	out_cfg ( 	OUT_23_DOH,
					para_s.DOH_Debounce_s16,
					f_100Hz_DU16,
					DOH_RESISTANCE_MIN,
					DOH_RESISTANCE_MAX );

	out_cfg ( 	OUT_24_DOH,
					para_s.DOH_Debounce_s16,
					f_100Hz_DU16,
					DOH_RESISTANCE_MIN,
					DOH_RESISTANCE_MAX );

	out_cfg ( 	OUT_25_DOH,
					para_s.DOH_Debounce_s16,
					f_100Hz_DU16,
					DOH_RESISTANCE_MIN,
					DOH_RESISTANCE_MAX );

	out_cfg ( 	OUT_26_DOH,
					para_s.DOH_Debounce_s16,
					f_100Hz_DU16,
					DOH_RESISTANCE_MIN,
					DOH_RESISTANCE_MAX );

	out_cfg ( 	OUT_27_DOH,
					para_s.DOH_Debounce_s16,
					f_100Hz_DU16,
					DOH_RESISTANCE_MIN,
					DOH_RESISTANCE_MAX );

	out_cfg ( 	OUT_28_DOH,
					para_s.DOH_Debounce_s16,
					f_100Hz_DU16,
					DOH_RESISTANCE_MIN,
					DOH_RESISTANCE_MAX );

	out_cfg ( 	OUT_29_DOH,
					para_s.DOH_Debounce_s16,
					f_100Hz_DU16,
					DOH_RESISTANCE_MIN,
					DOH_RESISTANCE_MAX );

	out_cfg ( 	OUT_30_DOH,
					para_s.DOH_Debounce_s16,
					f_100Hz_DU16,
					DOH_RESISTANCE_MIN,
					DOH_RESISTANCE_MAX );

	out_cfg ( 	OUT_31_DOH,
					para_s.DOH_Debounce_s16,
					f_100Hz_DU16,
					DOH_RESISTANCE_MIN,
					DOH_RESISTANCE_MAX );

	out_cfg ( 	OUT_32_DOH,
					para_s.DOH_Debounce_s16,
					f_100Hz_DU16,
					DOH_RESISTANCE_MIN,
					DOH_RESISTANCE_MAX );

(******************************************************************************************************)
(* Analog Output Voltage *)
(******************************************************************************************************)

IF para_s.Out_Cfg_33_s16 = PWM_MODE THEN
	out_cfg	(	OUT_33_POH,							(* PWM output close loop *)
					para_s.AOV_Debounce_s16,		(* debounce time [ms] for error detection *)
					para_s.AOC_Freq_s16, 			(* dither frequency [Hz] *)
					AOV_RESISTANCE_MIN, 				(* min resistance of solenoid for error detection [mOhm]*)
					AOV_RESISTANCE_MAX );			(* max resistance of solenoid for error detection[mOhm] *)

ELSIF para_s.Out_Cfg_33_s16 = AOV_MODE THEN
	out_cfg	(	OUT_33_AOV,							(* PWM output close loop *)
					para_s.AOV_Debounce_s16,		(* debounce time [ms] for error detection *)
					para_s.AOC_Freq_s16, 			(* dither frequency [Hz] *)
					AOV_RESISTANCE_MIN, 				(* min resistance of solenoid for error detection [mOhm]*)
					AOV_RESISTANCE_MAX );			(* max resistance of solenoid for error detection[mOhm] *)

	out_cfgPI(	OUT_33_AOV,							(*Channel*)
			      para_s.AOV_Kp_s16,				(*Kp factor*)
	      		para_s.AOV_Ki_s16 );				(*Ki factor*)
END_IF

IF para_s.Out_Cfg_34_s16 = PWM_MODE THEN
	out_cfg	(	OUT_34_POH,							(* PWM output close loop *)
					para_s.AOV_Debounce_s16,		(* debounce time [ms] for error detection *)
					para_s.AOC_Freq_s16, 			(* dither frequency [Hz] *)
					AOV_RESISTANCE_MIN, 				(* min resistance of solenoid for error detection [mOhm]*)
					AOV_RESISTANCE_MAX );			(* max resistance of solenoid for error detection[mOhm] *)

ELSIF para_s.Out_Cfg_34_s16 = AOV_MODE THEN
	out_cfg	(	OUT_34_AOV,							(* PWM output close loop *)
					para_s.AOV_Debounce_s16,		(* debounce time [ms] for error detection *)
					para_s.AOC_Freq_s16, 			(* dither frequency [Hz] *)
					AOV_RESISTANCE_MIN, 				(* min resistance of solenoid for error detection [mOhm]*)
					AOV_RESISTANCE_MAX );			(* max resistance of solenoid for error detection[mOhm] *)

	out_cfgPI(	OUT_34_AOV,							(*Channel*)
			      para_s.AOV_Kp_s16,				(*Kp factor*)
	      		para_s.AOV_Ki_s16 );				(*Ki factor*)
END_IF

IF para_s.Out_Cfg_35_s16 = PWM_MODE THEN
	out_cfg	(	OUT_35_POH,							(* PWM output close loop *)
					para_s.AOV_Debounce_s16,		(* debounce time [ms] for error detection *)
					para_s.AOC_Freq_s16, 			(* dither frequency [Hz] *)
					AOV_RESISTANCE_MIN, 				(* min resistance of solenoid for error detection [mOhm]*)
					AOV_RESISTANCE_MAX );			(* max resistance of solenoid for error detection[mOhm] *)

ELSIF para_s.Out_Cfg_35_s16 = AOV_MODE THEN
	out_cfg	(	OUT_35_AOV,							(* PWM output close loop *)
					para_s.AOV_Debounce_s16,		(* debounce time [ms] for error detection *)
					para_s.AOC_Freq_s16, 			(* dither frequency [Hz] *)
					AOV_RESISTANCE_MIN, 				(* min resistance of solenoid for error detection [mOhm]*)
					AOV_RESISTANCE_MAX );			(* max resistance of solenoid for error detection[mOhm] *)

	out_cfgPI(	OUT_35_AOV,							(*Channel*)
			      para_s.AOV_Kp_s16,				(*Kp factor*)
	      		para_s.AOV_Ki_s16 );				(*Ki factor*)
END_IF

IF para_s.Out_Cfg_36_s16 = PWM_MODE THEN
	out_cfg	(	OUT_36_POH,							(* PWM output close loop *)
					para_s.AOV_Debounce_s16,		(* debounce time [ms] for error detection *)
					para_s.AOC_Freq_s16, 			(* dither frequency [Hz] *)
					AOV_RESISTANCE_MIN, 				(* min resistance of solenoid for error detection [mOhm]*)
					AOV_RESISTANCE_MAX );			(* max resistance of solenoid for error detection[mOhm] *)

ELSIF para_s.Out_Cfg_36_s16 = AOV_MODE THEN
	out_cfg	(	OUT_36_AOV,							(* PWM output close loop *)
					para_s.AOV_Debounce_s16,		(* debounce time [ms] for error detection *)
					para_s.AOC_Freq_s16, 			(* dither frequency [Hz] *)
					AOV_RESISTANCE_MIN, 				(* min resistance of solenoid for error detection [mOhm]*)
					AOV_RESISTANCE_MAX );			(* max resistance of solenoid for error detection[mOhm] *)

	out_cfgPI(	OUT_36_AOV,							(*Channel*)
			      para_s.AOV_Kp_s16,				(*Kp factor*)
	      		para_s.AOV_Ki_s16 );				(*Ki factor*)
END_IF


(******************************************************************************************************)
(* Proportional Output Low *)
(******************************************************************************************************)
IF para_s.Out_Cfg_37_s16 = PWM_MODE THEN
	out_cfg	(	OUT_37_POL,							(* PWM output close loop *)
					para_s.POL_Debounce_s16,		(* debounce time [ms] for error detection *)
					POL_CL_DITHER_FREQUENCY, 		(* dither frequency [Hz] *)
					POL_CL_RESISTANCE_MIN, 			(* min resistance of solenoid for error detection [mOhm]*)
					POL_CL_RESISTANCE_MAX );		(* max resistance of solenoid for error detection[mOhm] *)
ELSIF para_s.Out_Cfg_37_s16 = PWM_CURRENT_MODE THEN
	out_cfg	(	OUT_37_POL_CL,						(* PWM output close loop *)
					para_s.POL_Debounce_s16,		(* debounce time [ms] for error detection *)
					POL_CL_DITHER_FREQUENCY, 		(* dither frequency [Hz] *)
					POL_CL_RESISTANCE_MIN, 			(* min resistance of solenoid for error detection [mOhm]*)
					POL_CL_RESISTANCE_MAX );		(* max resistance of solenoid for error detection[mOhm] *)

	out_cfgPI(	OUT_37_POL_CL,						(*Channel*)
			      para_s.POL_Kp_s16,				(*Kp factor*)
	      		para_s.POL_Ki_s16 );				(*Ki factor*)
END_IF

IF para_s.Out_Cfg_38_s16 = PWM_MODE THEN
	out_cfg	(	OUT_38_POL,							(* PWM output close loop *)
					para_s.POL_Debounce_s16,		(* debounce time [ms] for error detection *)
					POL_CL_DITHER_FREQUENCY, 		(* dither frequency [Hz] *)
					POL_CL_RESISTANCE_MIN, 			(* min resistance of solenoid for error detection [mOhm]*)
					POL_CL_RESISTANCE_MAX );		(* max resistance of solenoid for error detection[mOhm] *)
ELSIF para_s.Out_Cfg_38_s16 = PWM_CURRENT_MODE THEN
	out_cfg	(	OUT_38_POL_CL,						(* PWM output close loop *)
					para_s.POL_Debounce_s16,		(* debounce time [ms] for error detection *)
					POL_CL_DITHER_FREQUENCY, 		(* dither frequency [Hz] *)
					POL_CL_RESISTANCE_MIN, 			(* min resistance of solenoid for error detection [mOhm]*)
					POL_CL_RESISTANCE_MAX );		(* max resistance of solenoid for error detection[mOhm] *)

	out_cfgPI(	OUT_38_POL_CL,						(*Channel*)
			      para_s.POL_Kp_s16,				(*Kp factor*)
	      		para_s.POL_Ki_s16 );				(*Ki factor*)
END_IF

IF para_s.Out_Cfg_39_s16 = PWM_MODE THEN
	out_cfg	(	OUT_39_POL,							(* PWM output close loop *)
					para_s.POL_Debounce_s16,		(* debounce time [ms] for error detection *)
					POL_CL_DITHER_FREQUENCY, 		(* dither frequency [Hz] *)
					POL_CL_RESISTANCE_MIN, 			(* min resistance of solenoid for error detection [mOhm]*)
					POL_CL_RESISTANCE_MAX );		(* max resistance of solenoid for error detection[mOhm] *)
ELSIF para_s.Out_Cfg_39_s16 = PWM_CURRENT_MODE THEN
	out_cfg	(	OUT_39_POL_CL,						(* PWM output close loop *)
					para_s.POL_Debounce_s16,		(* debounce time [ms] for error detection *)
					POL_CL_DITHER_FREQUENCY, 		(* dither frequency [Hz] *)
					POL_CL_RESISTANCE_MIN, 			(* min resistance of solenoid for error detection [mOhm]*)
					POL_CL_RESISTANCE_MAX );		(* max resistance of solenoid for error detection[mOhm] *)

	out_cfgPI(	OUT_39_POL_CL,						(*Channel*)
			      para_s.POL_Kp_s16,				(*Kp factor*)
	      		para_s.POL_Ki_s16 );				(*Ki factor*)
END_IF

IF para_s.Out_Cfg_40_s16 = PWM_MODE THEN
	out_cfg	(	OUT_40_POL,							(* PWM output close loop *)
					para_s.POL_Debounce_s16,		(* debounce time [ms] for error detection *)
					POL_CL_DITHER_FREQUENCY, 		(* dither frequency [Hz] *)
					POL_CL_RESISTANCE_MIN, 			(* min resistance of solenoid for error detection [mOhm]*)
					POL_CL_RESISTANCE_MAX );		(* max resistance of solenoid for error detection[mOhm] *)
ELSIF para_s.Out_Cfg_40_s16 = PWM_CURRENT_MODE THEN
	out_cfg	(	OUT_40_POL_CL,						(* PWM output close loop *)
					para_s.POL_Debounce_s16,		(* debounce time [ms] for error detection *)
					POL_CL_DITHER_FREQUENCY, 		(* dither frequency [Hz] *)
					POL_CL_RESISTANCE_MIN, 			(* min resistance of solenoid for error detection [mOhm]*)
					POL_CL_RESISTANCE_MAX );		(* max resistance of solenoid for error detection[mOhm] *)

	out_cfgPI(	OUT_40_POL_CL,						(*Channel*)
			      para_s.POL_Kp_s16,				(*Kp factor*)
	      		para_s.POL_Ki_s16 );				(*Ki factor*)
END_IF

IF para_s.Out_Cfg_41_s16 = PWM_MODE THEN
	out_cfg	(	OUT_41_POL,							(* PWM output close loop *)
					para_s.POL_Debounce_s16,		(* debounce time [ms] for error detection *)
					POL_CL_DITHER_FREQUENCY, 		(* dither frequency [Hz] *)
					POL_CL_RESISTANCE_MIN, 			(* min resistance of solenoid for error detection [mOhm]*)
					POL_CL_RESISTANCE_MAX );		(* max resistance of solenoid for error detection[mOhm] *)
ELSIF para_s.Out_Cfg_41_s16 = PWM_CURRENT_MODE THEN
	out_cfg	(	OUT_41_POL_CL,						(* PWM output close loop *)
					para_s.POL_Debounce_s16,		(* debounce time [ms] for error detection *)
					POL_CL_DITHER_FREQUENCY, 		(* dither frequency [Hz] *)
					POL_CL_RESISTANCE_MIN, 			(* min resistance of solenoid for error detection [mOhm]*)
					POL_CL_RESISTANCE_MAX );		(* max resistance of solenoid for error detection[mOhm] *)

	out_cfgPI(	OUT_41_POL_CL,						(*Channel*)
			      para_s.POL_Kp_s16,				(*Kp factor*)
	      		para_s.POL_Ki_s16 );				(*Ki factor*)
END_IF

IF para_s.Out_Cfg_42_s16 = PWM_MODE THEN
	out_cfg	(	OUT_42_POL,							(* PWM output close loop *)
					para_s.POL_Debounce_s16,		(* debounce time [ms] for error detection *)
					POL_CL_DITHER_FREQUENCY, 		(* dither frequency [Hz] *)
					POL_CL_RESISTANCE_MIN, 			(* min resistance of solenoid for error detection [mOhm]*)
					POL_CL_RESISTANCE_MAX );		(* max resistance of solenoid for error detection[mOhm] *)
ELSIF para_s.Out_Cfg_42_s16 = PWM_CURRENT_MODE THEN
	out_cfg	(	OUT_42_POL_CL,						(* PWM output close loop *)
					para_s.POL_Debounce_s16,		(* debounce time [ms] for error detection *)
					POL_CL_DITHER_FREQUENCY, 		(* dither frequency [Hz] *)
					POL_CL_RESISTANCE_MIN, 			(* min resistance of solenoid for error detection [mOhm]*)
					POL_CL_RESISTANCE_MAX );		(* max resistance of solenoid for error detection[mOhm] *)

	out_cfgPI(	OUT_42_POL_CL,						(*Channel*)
			      para_s.POL_Kp_s16,				(*Kp factor*)
	      		para_s.POL_Ki_s16 );				(*Ki factor*)
END_IF

IF para_s.Out_Cfg_43_s16 = PWM_MODE THEN
	out_cfg	(	OUT_43_POL,							(* PWM output close loop *)
					para_s.POL_Debounce_s16,		(* debounce time [ms] for error detection *)
					POL_CL_DITHER_FREQUENCY, 		(* dither frequency [Hz] *)
					POL_CL_RESISTANCE_MIN, 			(* min resistance of solenoid for error detection [mOhm]*)
					POL_CL_RESISTANCE_MAX );		(* max resistance of solenoid for error detection[mOhm] *)
ELSIF para_s.Out_Cfg_43_s16 = PWM_CURRENT_MODE THEN
	out_cfg	(	OUT_43_POL_CL,						(* PWM output close loop *)
					para_s.POL_Debounce_s16,		(* debounce time [ms] for error detection *)
					POL_CL_DITHER_FREQUENCY, 		(* dither frequency [Hz] *)
					POL_CL_RESISTANCE_MIN, 			(* min resistance of solenoid for error detection [mOhm]*)
					POL_CL_RESISTANCE_MAX );		(* max resistance of solenoid for error detection[mOhm] *)

	out_cfgPI(	OUT_43_POL_CL,						(*Channel*)
			      para_s.POL_Kp_s16,				(*Kp factor*)
	      		para_s.POL_Ki_s16 );				(*Ki factor*)
END_IF

IF para_s.Out_Cfg_44_s16 = PWM_MODE THEN
	out_cfg	(	OUT_44_POL,							(* PWM output close loop *)
					para_s.POL_Debounce_s16,		(* debounce time [ms] for error detection *)
					POL_CL_DITHER_FREQUENCY, 		(* dither frequency [Hz] *)
					POL_CL_RESISTANCE_MIN, 			(* min resistance of solenoid for error detection [mOhm]*)
					POL_CL_RESISTANCE_MAX );		(* max resistance of solenoid for error detection[mOhm] *)
ELSIF para_s.Out_Cfg_44_s16 = PWM_CURRENT_MODE THEN
	out_cfg	(	OUT_44_POL_CL,						(* PWM output close loop *)
					para_s.POL_Debounce_s16,		(* debounce time [ms] for error detection *)
					POL_CL_DITHER_FREQUENCY, 		(* dither frequency [Hz] *)
					POL_CL_RESISTANCE_MIN, 			(* min resistance of solenoid for error detection [mOhm]*)
					POL_CL_RESISTANCE_MAX );		(* max resistance of solenoid for error detection[mOhm] *)

	out_cfgPI(	OUT_44_POL_CL,						(*Channel*)
			      para_s.POL_Kp_s16,				(*Kp factor*)
	      		para_s.POL_Ki_s16 );				(*Ki factor*)
END_IF

IF para_s.Out_Cfg_45_s16 = PWM_MODE THEN
	out_cfg	(	OUT_45_POL,							(* PWM output close loop *)
					para_s.POL_Debounce_s16,		(* debounce time [ms] for error detection *)
					POL_CL_DITHER_FREQUENCY, 		(* dither frequency [Hz] *)
					POL_CL_RESISTANCE_MIN, 			(* min resistance of solenoid for error detection [mOhm]*)
					POL_CL_RESISTANCE_MAX );		(* max resistance of solenoid for error detection[mOhm] *)
ELSIF para_s.Out_Cfg_45_s16 = PWM_CURRENT_MODE THEN
	out_cfg	(	OUT_45_POL_CL,						(* PWM output close loop *)
					para_s.POL_Debounce_s16,		(* debounce time [ms] for error detection *)
					POL_CL_DITHER_FREQUENCY, 		(* dither frequency [Hz] *)
					POL_CL_RESISTANCE_MIN, 			(* min resistance of solenoid for error detection [mOhm]*)
					POL_CL_RESISTANCE_MAX );		(* max resistance of solenoid for error detection[mOhm] *)

	out_cfgPI(	OUT_45_POL_CL,						(*Channel*)
			      para_s.POL_Kp_s16,				(*Kp factor*)
	      		para_s.POL_Ki_s16 );				(*Ki factor*)
END_IF

IF para_s.Out_Cfg_46_s16 = PWM_MODE THEN
	out_cfg	(	OUT_46_POL,							(* PWM output close loop *)
					para_s.POL_Debounce_s16,		(* debounce time [ms] for error detection *)
					POL_CL_DITHER_FREQUENCY, 		(* dither frequency [Hz] *)
					POL_CL_RESISTANCE_MIN, 			(* min resistance of solenoid for error detection [mOhm]*)
					POL_CL_RESISTANCE_MAX );		(* max resistance of solenoid for error detection[mOhm] *)
ELSIF para_s.Out_Cfg_46_s16 = PWM_CURRENT_MODE THEN
	out_cfg	(	OUT_46_POL_CL,						(* PWM output close loop *)
					para_s.POL_Debounce_s16,		(* debounce time [ms] for error detection *)
					POL_CL_DITHER_FREQUENCY, 		(* dither frequency [Hz] *)
					POL_CL_RESISTANCE_MIN, 			(* min resistance of solenoid for error detection [mOhm]*)
					POL_CL_RESISTANCE_MAX );		(* max resistance of solenoid for error detection[mOhm] *)

	out_cfgPI(	OUT_46_POL_CL,						(*Channel*)
			      para_s.POL_Kp_s16,				(*Kp factor*)
	      		para_s.POL_Ki_s16 );				(*Ki factor*)
END_IF


(******************************************************************************************************)
(* Analog Current Output *)
(******************************************************************************************************)

IF para_s.Out_Cfg_47_s16 = AOC_MODE THEN

	out_cfg (	OUT_47_AOC,
					para_s.AOC_Debounce_s16,
					para_s.AOC_Freq_s16,
					AOC_RESISTANCE_MIN,
					AOC_RESISTANCE_MAX);

	out_cfgPI(	OUT_47_AOC,							(*Channel*)
			      para_s.AOC_Kp_s16,				(*Kp factor*)
	      		para_s.AOC_Ki_s16 );				(*Ki factor*)
ELSIF para_s.Out_Cfg_47_s16 = AOV_MODE THEN
	out_cfg (	OUT_47_AOV,
					para_s.AOC_Debounce_s16,
					para_s.AOC_Freq_s16,
					AOC_RESISTANCE_MIN,
					AOC_RESISTANCE_MAX);

	out_cfgPI(	OUT_47_AOV,							(*Channel*)
			      para_s.AOC_Kp_s16,				(*Kp factor*)
	      		para_s.AOC_Ki_s16 );				(*Ki factor*)
END_IF

(*see API description for more explanations about the "min resistance" and "max resistance" parameters of the "out_cfg" function*)
END_ACTION
ACTION PLC_initCAN:
(*
!!! CAN1 always at 250kBaud !!!
!!! BODAS-service always on CAN1 !!!
!!! Databox No 1 and 2 are reserved by diagnosis !!!
!!! The first 20 databoxes of each CAN channel do not need a registration !!!
*)
(*can_setTxCycle(CAN_1, CAN1_MESSAGE_FREQ);*)
can_registerTxDataboxes(CAN_1, ADR(CAN_S.Data.can_TxMsg_as[1]), 42);
(*can_registerTxBuf(CAN_s.Chnl.ELOBAU_u8, ADR(CAN_s.Data.can_1_TxBuf_as[1]), 50);*)
(************************************************************************************************)
(******************** @CAN Initialization of CAN at 250kBaud ************************************)
(************************************************************************************************)

	can_cfgRxDatabox( CAN_s.Chnl.CAN_modem_u8,
							CAN_s.Box.Rx_Start_Stop_Button,
							CAN_s.Id.Rx_Start_Stop_Button,
							CAN_EXD_DU8		);


	can_cfgRxDatabox( CAN_s.Chnl.Remote_Control_u8,
							CAN_s.Box.Rx_RemoteControl_A_u16,
							CAN_s.Id.Rx_RemoteControl_A_u16,
							CAN_STD_DU8									);

	can_cfgRxDatabox( CAN_s.Chnl.Remote_Control_u8,
							CAN_s.Box.Rx_RemoteControl_B_u16,
						CAN_s.Id.Rx_RemoteControl_B_u16,
								CAN_STD_DU8									);

	can_cfgRxDatabox( CAN_s.Chnl.Remote_Control_u8,
							CAN_s.Box.Rx_RemoteControl_C_u16,
							CAN_s.Id.Rx_RemoteControl_C_u16,
							CAN_STD_DU8									);


	can_cfgRxDatabox( CAN_s.Chnl.Remote_Control_u8,
							CAN_s.Box.Rx_RemoteControl_C_u16,
							CAN_s.Id.Rx_RemoteControl_C_u16,
							CAN_STD_DU8									);

	can_cfgRxDatabox( CAN_1, 9, 16#18DA08F3, CAN_EXD_DU8);

		(*can_cfgTxDatabox(	CAN_s.Chnl.Remote_Control_u8,
								CAN_s.Box.Tx_Remote_Control_u16,
								CAN_s.Id.Tx_RemoteControl_u16,
								CAN_STD_DU8									);*)
(*END_IF*)
(***************************************************************************************************)
(***************************************************************************************************)
can_cfgRxDatabox( CAN_s.Chnl.CAN_modem_u8,
						CAN_s.Box.Rx_Modem_300,
						CAN_s.Id.Rx_Modem_300,
						CAN_EXD_DU8									);

can_cfgRxDatabox( CAN_s.Chnl.CAN_modem_u8,
						CAN_s.Box.Rx_Modem_301,
						CAN_s.Id.Rx_Modem_301,
						CAN_EXD_DU8									);


(***************************************************************************************************)

	can_cfgTxDatabox( CAN_1, 42, 16#18DAF308, CAN_EXD_DU8);

	can_cfgTxDatabox(	CAN_s.Chnl.CAN_modem_u8,
							CAN_s.Box.Tx_Modem_202,
							CAN_s.Id.Tx_Modem_202,
							CAN_EXD_DU8									);

	can_cfgTxDatabox(	CAN_s.Chnl.CAN_modem_u8,
							CAN_s.Box.Tx_Modem_203,
							CAN_s.Id.Tx_Modem_203,
							CAN_EXD_DU8									);

	can_cfgTxDatabox(	CAN_s.Chnl.CAN_modem_u8,
							CAN_s.Box.Tx_Modem_204,
							CAN_s.Id.Tx_Modem_204,
							CAN_EXD_DU8									);

	can_cfgTxDatabox(	CAN_s.Chnl.CAN_modem_u8,
							CAN_s.Box.Tx_Modem_205,
							CAN_s.Id.Tx_Modem_205,
							CAN_EXD_DU8									);

	can_cfgTxDatabox(	CAN_s.Chnl.CAN_modem_u8,
							CAN_s.Box.Tx_Modem_206,
							CAN_s.Id.Tx_Modem_206,
							CAN_EXD_DU8									);

	can_cfgTxDatabox(	CAN_s.Chnl.CAN_modem_u8,
							CAN_s.Box.Tx_Modem_207,
							CAN_s.Id.Tx_Modem_207,
							CAN_EXD_DU8									);

	can_cfgTxDatabox(	CAN_s.Chnl.CAN_modem_u8,
							CAN_s.Box.Tx_Modem_208,
							CAN_s.Id.Tx_Modem_208,
							CAN_EXD_DU8									);

	can_cfgTxDatabox(	CAN_s.Chnl.CAN_modem_u8,
							CAN_s.Box.Tx_Modem_209,
							CAN_s.Id.Tx_Modem_209,
							CAN_EXD_DU8									);

	can_cfgTxDatabox(	CAN_s.Chnl.CAN_modem_u8,
							CAN_s.Box.Tx_Modem_210,
							CAN_s.Id.Tx_Modem_210,
							CAN_EXD_DU8									);

	can_cfgTxDatabox(	CAN_s.Chnl.CAN_modem_u8,
							CAN_s.Box.Tx_Modem_211,
							CAN_s.Id.Tx_Modem_211,
							CAN_EXD_DU8									);

	can_cfgTxDatabox(	CAN_s.Chnl.CAN_modem_u8,
							CAN_s.Box.Tx_Modem_212,
							CAN_s.Id.Tx_Modem_212,
							CAN_EXD_DU8									);

	can_cfgTxDatabox(	CAN_s.Chnl.CAN_modem_u8,
							CAN_s.Box.Tx_Modem_213,
							CAN_s.Id.Tx_Modem_213,
							CAN_EXD_DU8									);

	can_cfgTxDatabox(	CAN_s.Chnl.CAN_modem_u8,
							CAN_s.Box.Tx_Modem_214,
							CAN_s.Id.Tx_Modem_214,
							CAN_EXD_DU8									);

	can_cfgTxDatabox(	CAN_s.Chnl.CAN_modem_u8,
							CAN_s.Box.Tx_Modem_215,
							CAN_s.Id.Tx_Modem_215,
							CAN_EXD_DU8									);

	can_cfgTxDatabox(	CAN_s.Chnl.CAN_modem_u8,
							CAN_s.Box.Tx_Modem_216,
							CAN_s.Id.Tx_Modem_216,
							CAN_EXD_DU8									);

	can_cfgTxDatabox(	CAN_s.Chnl.CAN_modem_u8,
							CAN_s.Box.Tx_MI3_220,
							CAN_s.Id.Tx_MI3_220,
							CAN_EXD_DU8									);

	can_cfgTxDatabox(	CAN_s.Chnl.CAN_modem_u8,
							CAN_s.Box.Tx_MI3_221,
							CAN_s.Id.Tx_MI3_221,
							CAN_EXD_DU8									);

	can_cfgTxDatabox(	CAN_s.Chnl.CAN_modem_u8,
							CAN_s.Box.Tx_Modem_303,
							CAN_s.Id.Tx_Modem_303,
							CAN_EXD_DU8									);

	can_cfgTxDatabox(	CAN_s.Chnl.CAN_modem_u8,
							CAN_s.Box.Tx_Modem_304,
							CAN_s.Id.Tx_Modem_304,
							CAN_EXD_DU8									);

	can_cfgTxDatabox(	CAN_s.Chnl.CAN_modem_u8,
							CAN_s.Box.Tx_Modem_305,
							CAN_s.Id.Tx_Modem_305,
							CAN_EXD_DU8									);

	can_cfgTxDatabox(	CAN_s.Chnl.CAN_modem_u8,
							CAN_s.Box.Tx_Modem_306,
							CAN_s.Id.Tx_Modem_306,
							CAN_EXD_DU8									);

	can_cfgTxDatabox(	CAN_s.Chnl.CAN_modem_u8,
							CAN_s.Box.Tx_Modem_307,
							CAN_s.Id.Tx_Modem_307,
							CAN_EXD_DU8									);

	can_cfgTxDatabox(	CAN_s.Chnl.CAN_modem_u8,
							CAN_s.Box.Tx_Modem_308,
							CAN_s.Id.Tx_Modem_308,
							CAN_EXD_DU8									);

	can_cfgTxDatabox(	CAN_s.Chnl.CAN_modem_u8,
							CAN_s.Box.Tx_Modem_309,
							CAN_s.Id.Tx_Modem_309,
							CAN_EXD_DU8									);

	can_cfgTxDatabox(	CAN_s.Chnl.CAN_modem_u8,
							CAN_s.Box.Tx_Modem_310,
							CAN_s.Id.Tx_Modem_310,
							CAN_EXD_DU8									);

	can_cfgTxDatabox(	CAN_s.Chnl.CAN_modem_u8,
							CAN_s.Box.Tx_Modem_311,
							CAN_s.Id.Tx_Modem_311,
							CAN_EXD_DU8									);

	can_cfgTxDatabox(	CAN_s.Chnl.CAN_modem_u8,
							CAN_s.Box.Tx_Modem_401,
							CAN_s.Id.Tx_Modem_401,
							CAN_EXD_DU8									);

	can_cfgTxDatabox(	CAN_s.Chnl.CAN_modem_u8,
							CAN_s.Box.Tx_Modem_402,
							CAN_s.Id.Tx_Modem_402,
							CAN_EXD_DU8									);

	can_cfgTxDatabox(	CAN_s.Chnl.CAN_modem_u8,
							CAN_s.Box.Tx_Modem_405,
							CAN_s.Id.Tx_Modem_405,
							CAN_EXD_DU8									);

	can_cfgTxDatabox(	CAN_s.Chnl.CAN_modem_u8,
							CAN_s.Box.Tx_Modem_406,
							CAN_s.Id.Tx_Modem_406,
							CAN_EXD_DU8									);

(*IF typeIndModule = DM_01 AND typeDieselSpSource	= CAN_TSC1 THEN*)
	can_cfgTxDatabox(	CAN_s.Chnl.CAN_modem_u8,
							CAN_s.Box.Tx_DM1_Diesel,
							CAN_s.Id.Tx_DM1_Diesel,
							CAN_EXD_DU8									);

	can_cfgTxDatabox(	CAN_s.Chnl.CAN_modem_u8,
							CAN_s.Box.Tx_DM2_Diesel,
							CAN_s.Id.Tx_DM2_Diesel,
							CAN_EXD_DU8									);

	can_cfgTxDatabox(	CAN_1,
							3,
							16#101,
							CAN_STD_DU8	);

(* Start CAN channel *)
can_init(CAN_1,	BAUD_250K);

	can_cfgTxDatabox(	CAN_2,
							3,
							16#102,
							CAN_STD_DU8	);

can_init(CAN_2,	BAUD_250K);

	can_cfgTxDatabox(	CAN_3,
							3,
							16#103,
							CAN_STD_DU8	);

can_init(CAN_3,	BAUD_250K);

	can_cfgTxDatabox(	CAN_4,
							3,
							16#104,
							CAN_STD_DU8	);

can_init(CAN_4,	BAUD_250K);
END_ACTION
ACTION PLC_initJ1939:
(************************************************************************************************)
(******************** @CAN Initialization of the databoxes to transmit **************************)
(************************************************************************************************)
(*CAN EASY functions are used. Be aware only 20 databoxes are supported*)
(*************************************************************************************************)
(********************************* Init J1939 - from API documentation ***************************)
(*************************************************************************************************)
 (* register can rx/tx buffers *)
  (*can_registerTxBuf(CAN_1, ADR(can1_tx_buf), 30); *)     (* not needed here !!! *)
  (*can_registerRxBuf(CAN_1, ADR(can1_rx_buf), 30); *)

  (* register j1939 rx/tx message boxes:
This FUNCTION registers memory FOR j1939 receive databoxes AND therefore defines the maximal number 
OF usable J1939 receive databoxes.

Remarks:
This function must be called once during the configuration of the J1939 communication stack before 
j1939_initComm(). After the execution of this function, each j1939 receive databox has to be 
initialized with j1939_initRxDatabox() before using. The meaning of this function is similar to 
the system function can_registerRxDataboxes().    *)

j1939_registerRxDataboxes( ADR(J1939_s.Data.j1939_RxMsg_as[1]), 8);
j1939_registerTxDataboxes( ADR(J1939_s.Data.j1939_TxMsg_as[1]), 20);

  (* Define j1939 receive messages within the j1939 RX databoxes: *)
  j1939_initRxDatabox(	J1939_s.Box.Rx_EEC1_u16,
								J1939_s.PGN.EEC1,
								J1939_s.SOURCE_ADRESS,
								J1939_s.TIMEOUT.EEC1,
								J1939_s.TIMEOUT.EEC1,
								J1939_s.Length.J1939_STD_MSG_LEN,
								ADR(J1939_s.Data.RxEEC1_au8[1]),
								J1939_s.DISABLE_CALLBACK				);

  j1939_initRxDatabox(	J1939_s.Box.Rx_ET1_u16,
								J1939_s.PGN.ET1_u32,
								J1939_s.SOURCE_ADRESS,
								J1939_s.TIMEOUT.ET1_u16,
								J1939_s.TIMEOUT.ET1_u16,
								J1939_s.Length.J1939_STD_MSG_LEN,
								ADR(J1939_s.Data.RxET1_au8[1]),
								J1939_s.DISABLE_CALLBACK				);

  j1939_initRxDatabox(	J1939_s.Box.Rx_EFL_u16,
								J1939_s.PGN.EFL_u32,
								J1939_s.SOURCE_ADRESS,
								J1939_s.TIMEOUT.EFL_u16,
								J1939_s.TIMEOUT.EFL_u16,
								J1939_s.Length.J1939_STD_MSG_LEN,
								ADR(J1939_s.Data.RxEFL_au8[1]),
								J1939_s.DISABLE_CALLBACK				);

  j1939_initRxDatabox(	J1939_s.Box.Rx_IC1_u16,
								J1939_s.PGN.IC1_u32,
								J1939_s.SOURCE_ADRESS,
								J1939_s.TIMEOUT.IC1_u16,
								J1939_s.TIMEOUT.IC1_u16,
								J1939_s.Length.J1939_STD_MSG_LEN,
								ADR(J1939_s.Data.RxIC1_au8[1]),
								J1939_s.DISABLE_CALLBACK				);

  j1939_initRxDatabox(	J1939_s.Box.Rx_DD_u16,
								J1939_s.PGN.DD,
								3,	(* Посылка не от двигателя *)
								J1939_s.TIMEOUT.DD_timeout,
								J1939_s.TIMEOUT.DD_timeout,
								J1939_s.Length.J1939_STD_MSG_LEN,
								ADR(J1939_s.Data.RxDD_au8[1]),
								J1939_s.DISABLE_CALLBACK				);

  (* Define j1939 receive messages within the j1939 RX databoxes: *)
  (*j1939_initRxDatabox(	J1939_s.Box.Rx_EEC2_u16,
								J1939_s.PGN.EEC2,
								J1939_s.SOURCE_ADRESS,
								J1939_s.TIMEOUT.EEC2,
								J1939_s.TIMEOUT.EEC2,
								J1939_s.Length.J1939_STD_MSG_LEN,
								ADR(J1939_s.Data.RxEEC2_au8[1]),
								J1939_s.DISABLE_CALLBACK				);

  (* Define j1939 receive messages within the j1939 RX databoxes: *)
  j1939_initRxDatabox(	J1939_s.Box.Rx_EEC3_u16,
								J1939_s.PGN.EEC3,
								J1939_s.SOURCE_ADRESS,
								J1939_s.TIMEOUT.EEC3,
								J1939_s.TIMEOUT.EEC3,
								J1939_s.Length.J1939_STD_MSG_LEN,
								ADR(J1939_s.Data.RxEEC3_au8[1]),
								J1939_s.DISABLE_CALLBACK				);*)

(*Tx***************************************************************************************************************)
(*********** 00 ************************************************************************)
	j1939_initTxDatabox(	J1939_s.Box.Tx_TF_u16,
   							J1939_s.PGN.TF_u32,
   							J1939_s.Length.PRIOR_DEFAULT, 		(* Prioritet *)
   							J1939_s.Length.CYCLE_DEFAULT,
   							J1939_s.Length.OFFSET_10,				(* offset *)
   							J1939_s.Length.J1939_STD_MSG_LEN, 	(* Length, byte *)
   							ADR( J1939_s.Data.TxTF_au8[1]),
   							J1939_s.DISABLE_CALLBACK				);
(*********** 01 ************************************************************************)
	j1939_initTxDatabox(	J1939_s.Box.Tx_ETC2_u16,
   							J1939_s.PGN.ETC2_u32,
   							J1939_s.Length.PRIOR_DEFAULT, 		(* Prioritet *)
   							J1939_s.Length.CYCLE_DEFAULT,
   							J1939_s.Length.OFFSET_10, 				(* offset *)
   							J1939_s.Length.J1939_STD_MSG_LEN, 	(* Length, byte *)
   							ADR( J1939_s.Data.TxETC2_au8[1]),
   							J1939_s.DISABLE_CALLBACK				);
(*********** 02 ************************************************************************)

(*********** 03 ************************************************************************)
	(*j1939_initTxDatabox(	J1939_S.Box.Tx_TFAC_u16,
								J1939_s.PGN.TFAC,
								J1939_s.Length.PRIOR_DEFAULT,
								J1939_s.Length.CYCLE_TFAC,
								J1939_s.Length.OFFSET_0,
								J1939_s.Length.J1939_STD_MSG_LEN,
								ADR(J1939_s.Data.TxTFAC_au8[1]),
								J1939_s.DISABLE_CALLBACK				);*)
(*********** 04 ************************************************************************)
	(*j1939_initTxDatabox(	J1939_s.Box.Tx_ETC2_u16,
   							J1939_s.PGN.ETC2_u32,
   							J1939_s.Length.PRIOR_DEFAULT,
								J1939_s.Length.CYCLE_DEFAULT,
								J1939_s.Length.OFFSET_0,
								J1939_s.Length.J1939_STD_MSG_LEN,
   							ADR( J1939_s.Data.TxETC2_au8[1]),
   							J1939_s.DISABLE_CALLBACK				);*)
(*********** 05 ************************************************************************)
	j1939_initTxDatabox(	J1939_s.Box.Tx_BJM1,
  	 							J1939_s.PGN.BJM1,
   							J1939_s.Length.PRIOR_DEFAULT,
								J1939_s.Length.CYCLE_LOCARUS,
								J1939_s.Length.OFFSET_10,
								J1939_s.Length.J1939_STD_MSG_LEN,
   							ADR( J1939_s.Data.TxBJM1[1]),
   							J1939_s.DISABLE_CALLBACK				);
(*********** 06 ************************************************************************)
	j1939_initTxDatabox(	J1939_s.Box.Tx_AV00MF,
  	 							J1939_s.PGN.AV00MF,
   							J1939_s.Length.PRIOR_DEFAULT,
								J1939_s.Length.CYCLE_LOCARUS,
								J1939_s.Length.OFFSET_20,
								J1939_s.Length.J1939_STD_MSG_LEN,
   							ADR( J1939_s.Data.TxAV00MF[1]),
   							J1939_s.DISABLE_CALLBACK				);
(*********** 07 ************************************************************************)
	j1939_initTxDatabox(	J1939_s.Box.Tx_AV01MF,
  	 							J1939_s.PGN.AV01MF,
   							J1939_s.Length.PRIOR_DEFAULT,
								J1939_s.Length.CYCLE_LOCARUS,
								J1939_s.Length.OFFSET_20,
								J1939_s.Length.J1939_STD_MSG_LEN,
   							ADR( J1939_s.Data.TxAV01MF[1]),
   							J1939_s.DISABLE_CALLBACK				);
(*********** 08 ************************************************************************)
	j1939_initTxDatabox(	J1939_s.Box.Tx_VF,
  	 							J1939_s.PGN.VF,
   							J1939_s.Length.PRIOR_DEFAULT,
								J1939_s.Length.CYCLE_LOCARUS,
								J1939_s.Length.OFFSET_0,
								J1939_s.Length.J1939_STD_MSG_LEN,
   							ADR( J1939_s.Data.TxVF[1]),
   							J1939_s.DISABLE_CALLBACK				);
(*********** 09 ************************************************************************)
	j1939_initTxDatabox(	J1939_s.Box.Tx_TRF2,
  	 							J1939_s.PGN.TRF2,
   							J1939_s.Length.PRIOR_DEFAULT,
								J1939_s.Length.CYCLE_LOCARUS,
								J1939_s.Length.OFFSET_0,
								J1939_s.Length.J1939_STD_MSG_LEN,
   							ADR( J1939_s.Data.TxTRF2[1]),
   							J1939_s.DISABLE_CALLBACK				);
(*********** 10 ************************************************************************)
	j1939_initTxDatabox(	J1939_s.Box.Tx_MP,
  	 							J1939_s.PGN.MP,
   							J1939_s.Length.PRIOR_DEFAULT,
								J1939_s.Length.CYCLE_LOCARUS,
								J1939_s.Length.OFFSET_0,
								J1939_s.Length.J1939_STD_MSG_LEN,
   							ADR( J1939_s.Data.TxMP[1]),
   							J1939_s.DISABLE_CALLBACK				);
(*********** 11 ************************************************************************)
	j1939_initTxDatabox(	J1939_s.Box.Tx_HOURS,
  	 							J1939_s.PGN.HOURS,
   							J1939_s.Length.PRIOR_DEFAULT,
								J1939_s.Length.CYCLE_LOCARUS,
								J1939_s.Length.OFFSET_0,
								J1939_s.Length.J1939_STD_MSG_LEN,
   							ADR( J1939_s.Data.TxHOURS[1]),
   							J1939_s.DISABLE_CALLBACK				);
(*********** 12-13 ************************************************************************)
(*********** 14 ************************************************************************)
	j1939_initTxDatabox(	J1939_s.Box.Tx_ESSI,
  	 							J1939_s.PGN.ESSI,
   							J1939_s.Length.PRIOR_DEFAULT,
								J1939_s.Length.CYCLE_LOCARUS,
								J1939_s.Length.OFFSET_0,
								J1939_s.Length.J1939_STD_MSG_LEN,
   							ADR( J1939_s.Data.TxESSI[1]),
   							J1939_s.DISABLE_CALLBACK				);
(*********** 15 ************************************************************************)
	j1939_initTxDatabox(	J1939_s.Box.Tx_AV02MF,
  	 							J1939_s.PGN.AV02MF,
   							J1939_s.Length.PRIOR_DEFAULT,
								J1939_s.Length.CYCLE_LOCARUS,
								J1939_s.Length.OFFSET_20,
								J1939_s.Length.J1939_STD_MSG_LEN,
   							ADR( J1939_s.Data.TxAV02MF[1]),
   							J1939_s.DISABLE_CALLBACK				);
(*********** 16 ************************************************************************)
	j1939_initTxDatabox(	J1939_s.Box.Tx_AV03MF,
  	 							J1939_s.PGN.AV03MF,
   							J1939_s.Length.PRIOR_DEFAULT,
								J1939_s.Length.CYCLE_LOCARUS,
								J1939_s.Length.OFFSET_20,
								J1939_s.Length.J1939_STD_MSG_LEN,
   							ADR( J1939_s.Data.TxAV03MF[1]),
   							J1939_s.DISABLE_CALLBACK				);
(*********** 17 ************************************************************************)
	j1939_initTxDatabox(	J1939_s.Box.Tx_AV04MF,
  	 							J1939_s.PGN.AV04MF,
   							J1939_s.Length.PRIOR_DEFAULT,
								J1939_s.Length.CYCLE_LOCARUS,
								J1939_s.Length.OFFSET_20,
								J1939_s.Length.J1939_STD_MSG_LEN,
   							ADR( J1939_s.Data.TxAV04MF[1]),
   							J1939_s.DISABLE_CALLBACK				);
(*********** 18 ************************************************************************)
	j1939_initTxDatabox(	J1939_s.Box.Tx_RHS,
  	 							J1939_s.PGN.RHS,
   							J1939_s.Length.PRIOR_DEFAULT,
								J1939_s.Length.CYCLE_LOCARUS,
								J1939_s.Length.OFFSET_10,
								J1939_s.Length.J1939_STD_MSG_LEN,
   							ADR( J1939_s.Data.TxRHS[1]),
   							J1939_s.DISABLE_CALLBACK				);
(*********** 19 ************************************************************************)
	j1939_initTxDatabox(	J1939_s.Box.Tx_LOI,
  	 							J1939_s.PGN.LOI,
   							J1939_s.Length.PRIOR_DEFAULT,
								J1939_s.Length.CYCLE_LOCARUS,
								J1939_s.Length.OFFSET_10,
								J1939_s.Length.J1939_STD_MSG_LEN,
   							ADR( J1939_s.Data.TxLOI[1]),
   							J1939_s.DISABLE_CALLBACK				);
(*********** Rx7 ************************************************************************)
  (* init a DM1 failure list for the DIESEL ECU with the address 00 *)
  j1939_initDiagnostic(	J1939_s.SOURCE_ADRESS,      			(* address of another ECU *)
                       	J1939_LIST_DM1_DU16,        			(* selected DM type = DM1 *)
                       	ADR(j1939_DIESEL_DM1_s),    			(* pointer to the failure list *)
                       	J1939_s.Box.Rx_DIESEL_DM1_u16, 		(* RX box nbr for receiving the list *)
                       	J1939_s.DISABLE_CALLBACK			); (* callback to evaluate failure *)
(*********** Rx8 ************************************************************************)
  (* init a DM2 failure list for the DIESEL ECU with the address 00 *)
  j1939_initDiagnostic(	J1939_s.SOURCE_ADRESS,      			(* address of another ECU *)
                       	J1939_LIST_DM2_DU16,        			(* selected DM type = DM1 *)
                       	ADR(j1939_DIESEL_DM2_s),    			(* pointer to the failure list *)
                       	J1939_s.Box.Rx_DIESEL_DM2_u16, 		(* RX box nbr for receiving the list *)
                       	J1939_s.DISABLE_CALLBACK			); (* callback to evaluate failure *)
(***************************************************************************************)
	(* define the controller application name, required for address claiming *)
  j1939_setCaName(16#02,  (* 3 bit industry group *)
                  16#00,  (* 4 bit vehicle instance *)
                  16#01,  (* 7 bit vehicle system *)
                  16#81,  (* 8 bit function *)
                  16#01,  (* 5 bit function instance *)
                  16#01); (* 3 bit ecu instance *)

  (* initialize and start j1939 communication *)
  j1939_initComm(				CAN_s.Chnl.J1939_DIESEL_u8,
									16#03, 								(* RC controllrer own address *)
									100,  								(*	Priority OF the j1939 task, not used in BodasDesign*)
									CYCLE,
									20);									(* Maximum allowed run time of the j1939 task,
																				related to the J1939 cycle time, %%, [1...99] *)
(***************************************************************************************)
END_ACTION

(* POU Callback_MAIN_Task, SFC *)
	PROGRAM Callback_MAIN_Task
VAR
	Mo_ErrorCheck_Ignore_b8				: BOOL;
	Mo_ErrorCheck_LimpHome_b8			: BOOL;
	Mo_ErrorCheck_Stop_b8				: BOOL;
	Mo_ErrorCheck_Switch_b8				: BOOL;
(*	stError_dw: DWORD;*)  (*VL: all start errors are in "err" structure*)
	stCase_u16								: UINT; (* Statemachine of the Startlock *)
	LC_Done_b8								: BOOL := FALSE;
	FirstCycle_b8							: BOOL := TRUE;
	calc_Diesel_Poti_Ramp_fb			: mat_calcRamp;
	counter									: INT				:= 0;
	VAR1										: DINT := 17;
	VAR2										: DINT := 16#1A;
END_VAR
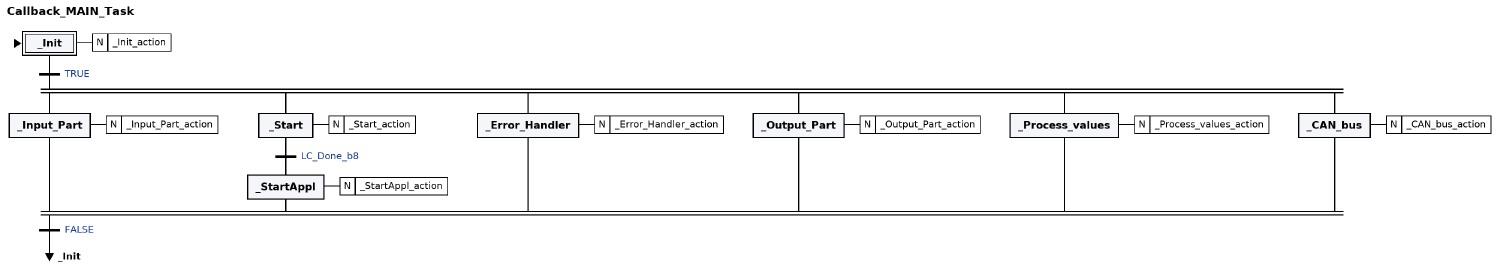
INITIAL_STEP _Init:
	_Init_action(N);
END_STEP
TRANSITION FROM _Init TO (_Input_Part, _Start, _Error_Handler, _Output_Part, _Process_values, _CAN_bus) := TRUE;
END_TRANSITION
STEP _Input_Part:
	_Input_Part_action(N);
END_STEP
STEP _Start:
	_Start_action(N);
END_STEP
TRANSITION FROM _Start TO _StartAppl := LC_Done_b8;
END_TRANSITION
STEP _StartAppl:
	_StartAppl_action(N);
END_STEP
STEP _Error_Handler:
	_Error_Handler_action(N);
END_STEP
STEP _Output_Part:
	_Output_Part_action(N);
END_STEP
STEP _Process_values:
	_Process_values_action(N);
END_STEP
STEP _CAN_bus:
	_CAN_bus_action(N);
END_STEP
TRANSITION FROM (_Input_Part, _StartAppl, _Error_Handler, _Output_Part, _Process_values, _CAN_bus) TO _Init := FALSE;
END_TRANSITION

ACTION _Init_action:
sys_triggerTC(PLC_PRG.MAIN_Task_Handle_u8);
END_ACTION

ACTION _Input_Part_action:
sys_triggerTC(PLC_PRG.MAIN_Task_Handle_u8);


Get_System_Info();			(* *)
(*Get_Dig_Freq_Inputs();		(* *)*)

get_Status();
END_ACTION

ACTION _Start_action:
(***********************************************************************************)
(******************** Start lock  **************************************************)
(***********************************************************************************)

Startlock_RC28_14(
	StartconditionAppl_I_b8		:= TRUE,
	StartconditionAppl_II_b8	:= TRUE,
	StartconditionEngine_b8		:= TRUE,
(* All appl. start conditions after Learning Curve action *)
	EnableSafout_b8				:= TRUE,
	tiCycle_s16						:= CYCLE,
	Mo_ErrorCheck_Ignore_b8		=> Mo_ErrorCheck_Ignore_b8,
	Mo_ErrorCheck_LimpHome_b8	=> Mo_ErrorCheck_LimpHome_b8,
	Mo_ErrorCheck_Stop_b8		=> Mo_ErrorCheck_Stop_b8,
	Mo_ErrorCheck_Switch_b8		=> Mo_ErrorCheck_Switch_b8,
	stCase_u16 						=> stCase_u16
);

	stStartlock_b8 := Startlock_RC28_14.StartEnable_b8;
END_ACTION

ACTION _StartAppl_action:
stStartAppl_b8 := TRUE;
END_ACTION

ACTION _Error_Handler_action:
proc_Err_CAN();
proc_Err_DIG_outs();
proc_Err_Inputs();
proc_Err_Power();
proc_Err_PWM();
proc_Err_Sensors();
proc_Err_Status();
proc_Err_Parameters();

review_Errors(
	Saved_Err_b8:= FALSE,
	Last_Error_Shown_b8:= flash_Error_Code.Error_Indication_Completed_b8,
	Displayed_Err_Code_s16 => );

flash_Error_Code(
	BlinkCode_s16:= review_Errors.Displayed_Err_Code_s16,
	tiBlink10H_u32:= t#1s,
	tiBlink10L_u32:= t#500ms,
	tiBlinkPause_10_1_u32:= t#500ms,
	tiBlink1_H_u32:= t#500ms,
	tiBlink1_L_u32:= t#500ms,
	tiPauseLong_u32:= t#500ms,
	ErrLamp_b8=> (*output.set_lamp_Error_b8*),
	Error_Indication_Completed_b8=> );
END_ACTION

ACTION _Output_Part_action:
out_DIG();
out_Current();
out_Status();
out_Control();
END_ACTION

ACTION _Process_values_action:
diag_setProcessVar(0, 0, VAR1);
diag_setProcessVar(0, 1, 0);
diag_setProcessVar(0, 2, 0);
diag_setProcessVar(0, 3, 0);
diag_setProcessVar(0, 4, SW_Version.SW_Git_Commit_s32);
diag_setProcessVar(0, 5, SW_Version.SW_Git_Commit_s32);
diag_setProcessVar(0, 6, SW_Version.SW_Git_Commit_s32);
diag_setProcessVar(0, 7, SW_Version.SW_Git_Commit_s32);

diag_setProcessVar(1, 0, VAR1);
diag_setProcessVar(1, 1, VAR2);
diag_setProcessVar(1, 2, 0);
diag_setProcessVar(1, 3, 0);
diag_setProcessVar(1, 4, 0);
diag_setProcessVar(1, 5, 0);
diag_setProcessVar(1, 6, 0);
diag_setProcessVar(1, 7, 0);

diag_setProcessVar(2, 0, 0);
diag_setProcessVar(2, 1, 0);
diag_setProcessVar(2, 2, 0);
diag_setProcessVar(2, 3, 0);
diag_setProcessVar(2, 4, 0);
diag_setProcessVar(2, 5, 0);
diag_setProcessVar(2, 6, 0);
diag_setProcessVar(2, 7, 0);

diag_setProcessVar(3, 0, 0);
diag_setProcessVar(3, 1, 0);
diag_setProcessVar(3, 2, 0);
diag_setProcessVar(3, 3, 0);
diag_setProcessVar(3, 4, 0);
diag_setProcessVar(3, 5, 0);
diag_setProcessVar(3, 6, 0);
diag_setProcessVar(3, 7, 0);

diag_setProcessVar(4, 0, 0);
diag_setProcessVar(4, 1, 0);
diag_setProcessVar(4, 2, 0);
diag_setProcessVar(4, 3, 0);
diag_setProcessVar(4, 4, 0);
diag_setProcessVar(4, 5, 0);
diag_setProcessVar(4, 6, 0);
diag_setProcessVar(4, 7, 0);

(*****************************************************************************)
diag_setProcessVar(5, 0, 0);
diag_setProcessVar(5, 1, 0);
diag_setProcessVar(5, 2, 0);
diag_setProcessVar(5, 3, 0);
diag_setProcessVar(5, 4, 0);
diag_setProcessVar(5, 5, 0);
diag_setProcessVar(5, 6, 0);
diag_setProcessVar(5, 7, 0);

diag_setProcessVar(6, 0, 0);
diag_setProcessVar(6, 1, 0);
diag_setProcessVar(6, 2, 0);
diag_setProcessVar(6, 3, 0);
diag_setProcessVar(6, 4, 0);
diag_setProcessVar(6, 5, 0);
diag_setProcessVar(6, 6, 0);
diag_setProcessVar(6, 7, 0);

diag_setProcessVar(7, 0, 0);
diag_setProcessVar(7, 1, 0);
diag_setProcessVar(7, 2, 0);
diag_setProcessVar(7, 3, 0);
diag_setProcessVar(7, 4, 0);
diag_setProcessVar(7, 5, 0);
diag_setProcessVar(7, 6, 0);
diag_setProcessVar(7, 7, 0);

diag_setProcessVar(8, 0, 0);
diag_setProcessVar(8, 1, 0);
diag_setProcessVar(8, 2, 0);
diag_setProcessVar(8, 3, 0);
diag_setProcessVar(8, 4, 0);
diag_setProcessVar(8, 5, 0);
diag_setProcessVar(8, 6, 0);
diag_setProcessVar(8, 7, 0);

diag_setProcessVar(9, 0, 0);
diag_setProcessVar(9, 1, 0);
diag_setProcessVar(9, 2, 0);
diag_setProcessVar(9, 3, 0);
diag_setProcessVar(9, 4, 0);
diag_setProcessVar(9, 5, 0);
diag_setProcessVar(9, 6, 0);
diag_setProcessVar(9, 7, 0);
(*****************************************************************************)
(*****************************************************************************)
(*****************************************************************************)
diag_setProcessVar(10, 0, 0);	(* input.tOil_degC_s16); 			*)
diag_setProcessVar(10, 1, 0);	(* input.tCoolant_DegC_s16);	*)
diag_setProcessVar(10, 2, 0);
diag_setProcessVar(10, 3, 0);
diag_setProcessVar(10, 4, 0);
diag_setProcessVar(10, 5, 0);
diag_setProcessVar(10, 6, 0);
diag_setProcessVar(10, 7, 0);


diag_setProcessVar(23, 0, get_Status.in_as[1].in_aiv_s.u_mV_u16);	(* input.tOil_degC_s16); 			*)
diag_setProcessVar(23, 1, get_Status.in_as[1].in_aiv_s.diag_u8);	(* input.tCoolant_DegC_s16);	*)
diag_setProcessVar(23, 2, get_Status.in_as[1].in_aiv_s.diagDebounced_u8);
diag_setProcessVar(23, 3, get_Status.in_as[1].in_aiv_s.digits_u16);
diag_setProcessVar(23, 4, BOOL_TO_INT(get_Status.in_as[1].in_aiv_s.state_l));
diag_setProcessVar(23, 5, BOOL_TO_INT(get_Status.in_as[1].in_aiv_s.stateDebounced_l));
diag_setProcessVar(23, 6, get_Status.in_as[1].in_aiv_s.status_b16);
diag_setProcessVar(23, 7, para_s.Out_Val_01_s16);


diag_setProcessVar(31, 0, get_Status.in_as[1].in_aiv_s.u_mV_u16);	(* input.tOil_degC_s16); 			*)
diag_setProcessVar(31, 1, get_Status.in_as[1].in_aiv_s.diag_u8);	(* input.tCoolant_DegC_s16);	*)
diag_setProcessVar(31, 2, get_Status.in_as[1].in_aiv_s.diagDebounced_u8);
diag_setProcessVar(31, 3, get_Status.in_as[1].in_aiv_s.digits_u16);
diag_setProcessVar(31, 4, BOOL_TO_INT(get_Status.in_as[1].in_aiv_s.state_l));
diag_setProcessVar(31, 5, BOOL_TO_INT(get_Status.in_as[1].in_aiv_s.stateDebounced_l));
diag_setProcessVar(31, 6, get_Status.in_as[1].in_aiv_s.status_b16);
diag_setProcessVar(31, 7, para_s.Out_Val_01_s16);

diag_setProcessVar(32, 0, get_Status.in_as[1].in_aiv_s.u_mV_u16);	(* input.tOil_degC_s16); 			*)
diag_setProcessVar(32, 1, get_Status.in_as[1].in_aiv_s.diag_u8);	(* input.tCoolant_DegC_s16);	*)
diag_setProcessVar(32, 2, get_Status.in_as[1].in_aiv_s.diagDebounced_u8);
diag_setProcessVar(32, 3, get_Status.in_as[1].in_aiv_s.digits_u16);
diag_setProcessVar(32, 4, BOOL_TO_INT(get_Status.in_as[1].in_aiv_s.state_l));
diag_setProcessVar(32, 5, BOOL_TO_INT(get_Status.in_as[1].in_aiv_s.stateDebounced_l));
diag_setProcessVar(32, 6, get_Status.in_as[1].in_aiv_s.status_b16);
diag_setProcessVar(32, 7, para_s.Out_Val_01_s16);

diag_setProcessVar(33, 0, get_Status.in_as[1].in_aiv_s.u_mV_u16);	(* input.tOil_degC_s16); 			*)
diag_setProcessVar(33, 1, get_Status.in_as[1].in_aiv_s.diag_u8);	(* input.tCoolant_DegC_s16);	*)
diag_setProcessVar(33, 2, get_Status.in_as[1].in_aiv_s.diagDebounced_u8);
diag_setProcessVar(33, 3, get_Status.in_as[1].in_aiv_s.digits_u16);
diag_setProcessVar(33, 4, BOOL_TO_INT(get_Status.in_as[1].in_aiv_s.state_l));
diag_setProcessVar(33, 5, BOOL_TO_INT(get_Status.in_as[1].in_aiv_s.stateDebounced_l));
diag_setProcessVar(33, 6, get_Status.in_as[1].in_aiv_s.status_b16);
diag_setProcessVar(33, 7, para_s.Out_Val_01_s16);

diag_setProcessVar(34, 0, get_Status.in_as[1].in_aiv_s.u_mV_u16);	(* input.tOil_degC_s16); 			*)
diag_setProcessVar(34, 1, get_Status.in_as[1].in_aiv_s.diag_u8);	(* input.tCoolant_DegC_s16);	*)
diag_setProcessVar(34, 2, get_Status.in_as[1].in_aiv_s.diagDebounced_u8);
diag_setProcessVar(34, 3, get_Status.in_as[1].in_aiv_s.digits_u16);
diag_setProcessVar(34, 4, BOOL_TO_INT(get_Status.in_as[1].in_aiv_s.state_l));
diag_setProcessVar(34, 5, BOOL_TO_INT(get_Status.in_as[1].in_aiv_s.stateDebounced_l));
diag_setProcessVar(34, 6, get_Status.in_as[1].in_aiv_s.status_b16);
diag_setProcessVar(34, 7, para_s.Out_Val_01_s16);

diag_setProcessVar(35, 0, get_Status.in_as[1].in_aiv_s.u_mV_u16);	(* input.tOil_degC_s16); 			*)
diag_setProcessVar(35, 1, get_Status.in_as[1].in_aiv_s.diag_u8);	(* input.tCoolant_DegC_s16);	*)
diag_setProcessVar(35, 2, get_Status.in_as[1].in_aiv_s.diagDebounced_u8);
diag_setProcessVar(35, 3, get_Status.in_as[1].in_aiv_s.digits_u16);
diag_setProcessVar(35, 4, BOOL_TO_INT(get_Status.in_as[1].in_aiv_s.state_l));
diag_setProcessVar(35, 5, BOOL_TO_INT(get_Status.in_as[1].in_aiv_s.stateDebounced_l));
diag_setProcessVar(35, 6, get_Status.in_as[1].in_aiv_s.status_b16);
diag_setProcessVar(35, 7, para_s.Out_Val_01_s16);

diag_setProcessVar(36, 0, get_Status.in_as[1].in_aiv_s.u_mV_u16);	(* input.tOil_degC_s16); 			*)
diag_setProcessVar(36, 1, get_Status.in_as[1].in_aiv_s.diag_u8);	(* input.tCoolant_DegC_s16);	*)
diag_setProcessVar(36, 2, get_Status.in_as[1].in_aiv_s.diagDebounced_u8);
diag_setProcessVar(36, 3, get_Status.in_as[1].in_aiv_s.digits_u16);
diag_setProcessVar(36, 4, BOOL_TO_INT(get_Status.in_as[1].in_aiv_s.state_l));
diag_setProcessVar(36, 5, BOOL_TO_INT(get_Status.in_as[1].in_aiv_s.stateDebounced_l));
diag_setProcessVar(36, 6, get_Status.in_as[1].in_aiv_s.status_b16);
diag_setProcessVar(36, 7, para_s.Out_Val_01_s16);

diag_setProcessVar(37, 0, get_Status.in_as[1].in_aiv_s.u_mV_u16);	(* input.tOil_degC_s16); 			*)
diag_setProcessVar(37, 1, get_Status.in_as[1].in_aiv_s.diag_u8);	(* input.tCoolant_DegC_s16);	*)
diag_setProcessVar(37, 2, get_Status.in_as[1].in_aiv_s.diagDebounced_u8);
diag_setProcessVar(37, 3, get_Status.in_as[1].in_aiv_s.digits_u16);
diag_setProcessVar(37, 4, BOOL_TO_INT(get_Status.in_as[1].in_aiv_s.state_l));
diag_setProcessVar(37, 5, BOOL_TO_INT(get_Status.in_as[1].in_aiv_s.stateDebounced_l));
diag_setProcessVar(37, 6, get_Status.in_as[1].in_aiv_s.status_b16);
diag_setProcessVar(37, 7, para_s.Out_Val_01_s16);

diag_setProcessVar(38, 0, get_Status.in_as[1].in_aiv_s.u_mV_u16);	(* input.tOil_degC_s16); 			*)
diag_setProcessVar(38, 1, get_Status.in_as[1].in_aiv_s.diag_u8);	(* input.tCoolant_DegC_s16);	*)
diag_setProcessVar(38, 2, get_Status.in_as[1].in_aiv_s.diagDebounced_u8);
diag_setProcessVar(38, 3, get_Status.in_as[1].in_aiv_s.digits_u16);
diag_setProcessVar(38, 4, BOOL_TO_INT(get_Status.in_as[1].in_aiv_s.state_l));
diag_setProcessVar(38, 5, BOOL_TO_INT(get_Status.in_as[1].in_aiv_s.stateDebounced_l));
diag_setProcessVar(38, 6, get_Status.in_as[1].in_aiv_s.status_b16);
diag_setProcessVar(38, 7, para_s.Out_Val_01_s16);

diag_setProcessVar(39, 0, get_Status.in_as[1].in_aiv_s.u_mV_u16);	(* input.tOil_degC_s16); 			*)
diag_setProcessVar(39, 1, get_Status.in_as[1].in_aiv_s.diag_u8);	(* input.tCoolant_DegC_s16);	*)
diag_setProcessVar(39, 2, get_Status.in_as[1].in_aiv_s.diagDebounced_u8);
diag_setProcessVar(39, 3, get_Status.in_as[1].in_aiv_s.digits_u16);
diag_setProcessVar(39, 4, BOOL_TO_INT(get_Status.in_as[1].in_aiv_s.state_l));
diag_setProcessVar(39, 5, BOOL_TO_INT(get_Status.in_as[1].in_aiv_s.stateDebounced_l));
diag_setProcessVar(39, 6, get_Status.in_as[1].in_aiv_s.status_b16);
diag_setProcessVar(39, 7, para_s.Out_Val_01_s16);

diag_setProcessVar(40, 0, get_Status.in_as[1].in_aiv_s.u_mV_u16);	(* input.tOil_degC_s16); 			*)
diag_setProcessVar(40, 1, get_Status.in_as[1].in_aiv_s.diag_u8);	(* input.tCoolant_DegC_s16);	*)
diag_setProcessVar(40, 2, get_Status.in_as[1].in_aiv_s.diagDebounced_u8);
diag_setProcessVar(40, 3, get_Status.in_as[1].in_aiv_s.digits_u16);
diag_setProcessVar(40, 4, BOOL_TO_INT(get_Status.in_as[1].in_aiv_s.state_l));
diag_setProcessVar(40, 5, BOOL_TO_INT(get_Status.in_as[1].in_aiv_s.stateDebounced_l));
diag_setProcessVar(40, 6, get_Status.in_as[1].in_aiv_s.status_b16);
diag_setProcessVar(40, 7, para_s.Out_Val_01_s16);

diag_setProcessVar(41, 0, get_Status.in_as[1].in_aiv_s.u_mV_u16);	(* input.tOil_degC_s16); 			*)
diag_setProcessVar(41, 1, get_Status.in_as[1].in_aiv_s.diag_u8);	(* input.tCoolant_DegC_s16);	*)
diag_setProcessVar(41, 2, get_Status.in_as[1].in_aiv_s.diagDebounced_u8);
diag_setProcessVar(41, 3, get_Status.in_as[1].in_aiv_s.digits_u16);
diag_setProcessVar(41, 4, BOOL_TO_INT(get_Status.in_as[1].in_aiv_s.state_l));
diag_setProcessVar(41, 5, BOOL_TO_INT(get_Status.in_as[1].in_aiv_s.stateDebounced_l));
diag_setProcessVar(41, 6, get_Status.in_as[1].in_aiv_s.status_b16);
diag_setProcessVar(41, 7, para_s.Out_Val_01_s16);

diag_setProcessVar(42, 0, get_Status.in_as[1].in_aiv_s.u_mV_u16);	(* input.tOil_degC_s16); 			*)
diag_setProcessVar(42, 1, get_Status.in_as[1].in_aiv_s.diag_u8);	(* input.tCoolant_DegC_s16);	*)
diag_setProcessVar(42, 2, get_Status.in_as[1].in_aiv_s.diagDebounced_u8);
diag_setProcessVar(42, 3, get_Status.in_as[1].in_aiv_s.digits_u16);
diag_setProcessVar(42, 4, BOOL_TO_INT(get_Status.in_as[1].in_aiv_s.state_l));
diag_setProcessVar(42, 5, BOOL_TO_INT(get_Status.in_as[1].in_aiv_s.stateDebounced_l));
diag_setProcessVar(42, 6, get_Status.in_as[1].in_aiv_s.status_b16);
diag_setProcessVar(42, 7, para_s.Out_Val_01_s16);

diag_setProcessVar(43, 0, get_Status.in_as[1].in_aiv_s.u_mV_u16);	(* input.tOil_degC_s16); 			*)
diag_setProcessVar(43, 1, get_Status.in_as[1].in_aiv_s.diag_u8);	(* input.tCoolant_DegC_s16);	*)
diag_setProcessVar(43, 2, get_Status.in_as[1].in_aiv_s.diagDebounced_u8);
diag_setProcessVar(43, 3, get_Status.in_as[1].in_aiv_s.digits_u16);
diag_setProcessVar(43, 4, BOOL_TO_INT(get_Status.in_as[1].in_aiv_s.state_l));
diag_setProcessVar(43, 5, BOOL_TO_INT(get_Status.in_as[1].in_aiv_s.stateDebounced_l));
diag_setProcessVar(43, 6, get_Status.in_as[1].in_aiv_s.status_b16);
diag_setProcessVar(43, 7, para_s.Out_Val_01_s16);

diag_setProcessVar(44, 0, get_Status.in_as[1].in_aiv_s.u_mV_u16);	(* input.tOil_degC_s16); 			*)
diag_setProcessVar(44, 1, get_Status.in_as[1].in_aiv_s.diag_u8);	(* input.tCoolant_DegC_s16);	*)
diag_setProcessVar(44, 2, get_Status.in_as[1].in_aiv_s.diagDebounced_u8);
diag_setProcessVar(44, 3, get_Status.in_as[1].in_aiv_s.digits_u16);
diag_setProcessVar(44, 4, BOOL_TO_INT(get_Status.in_as[1].in_aiv_s.state_l));
diag_setProcessVar(44, 5, BOOL_TO_INT(get_Status.in_as[1].in_aiv_s.stateDebounced_l));
diag_setProcessVar(44, 6, get_Status.in_as[1].in_aiv_s.status_b16);
diag_setProcessVar(44, 7, para_s.Out_Val_01_s16);

diag_setProcessVar(45, 0, get_Status.in_as[1].in_aiv_s.u_mV_u16);	(* input.tOil_degC_s16); 			*)
diag_setProcessVar(45, 1, get_Status.in_as[1].in_aiv_s.diag_u8);	(* input.tCoolant_DegC_s16);	*)
diag_setProcessVar(45, 2, get_Status.in_as[1].in_aiv_s.diagDebounced_u8);
diag_setProcessVar(45, 3, get_Status.in_as[1].in_aiv_s.digits_u16);
diag_setProcessVar(45, 4, BOOL_TO_INT(get_Status.in_as[1].in_aiv_s.state_l));
diag_setProcessVar(45, 5, BOOL_TO_INT(get_Status.in_as[1].in_aiv_s.stateDebounced_l));
diag_setProcessVar(45, 6, get_Status.in_as[1].in_aiv_s.status_b16);
diag_setProcessVar(45, 7, para_s.Out_Val_01_s16);

diag_setProcessVar(46, 0, get_Status.in_as[1].in_aiv_s.u_mV_u16);	(* input.tOil_degC_s16); 			*)
diag_setProcessVar(46, 1, get_Status.in_as[1].in_aiv_s.diag_u8);	(* input.tCoolant_DegC_s16);	*)
diag_setProcessVar(46, 2, get_Status.in_as[1].in_aiv_s.diagDebounced_u8);
diag_setProcessVar(46, 3, get_Status.in_as[1].in_aiv_s.digits_u16);
diag_setProcessVar(46, 4, BOOL_TO_INT(get_Status.in_as[1].in_aiv_s.state_l));
diag_setProcessVar(46, 5, BOOL_TO_INT(get_Status.in_as[1].in_aiv_s.stateDebounced_l));
diag_setProcessVar(46, 6, get_Status.in_as[1].in_aiv_s.status_b16);
diag_setProcessVar(46, 7, para_s.Out_Val_01_s16);

diag_setProcessVar(47, 0, get_Status.in_as[1].in_aiv_s.u_mV_u16);	(* input.tOil_degC_s16); 			*)
diag_setProcessVar(47, 1, get_Status.in_as[1].in_aiv_s.diag_u8);	(* input.tCoolant_DegC_s16);	*)
diag_setProcessVar(47, 2, get_Status.in_as[1].in_aiv_s.diagDebounced_u8);
diag_setProcessVar(47, 3, get_Status.in_as[1].in_aiv_s.digits_u16);
diag_setProcessVar(47, 4, BOOL_TO_INT(get_Status.in_as[1].in_aiv_s.state_l));
diag_setProcessVar(47, 5, BOOL_TO_INT(get_Status.in_as[1].in_aiv_s.stateDebounced_l));
diag_setProcessVar(47, 6, get_Status.in_as[1].in_aiv_s.status_b16);
diag_setProcessVar(47, 7, para_s.Out_Val_01_s16);
END_ACTION

ACTION _CAN_bus_action:
(* status of CAN channel CAN_1 *)
CAN_s.Status.Channel_CAN_1 := can_getStatus(CAN_1);

CAN_s.Data.Databox_data_1[1] := INT_TO_USINT(counter);
CAN_s.Data.Databox_data_2[2] := INT_TO_USINT(counter);
CAN_s.Data.Databox_data_3[3] := INT_TO_USINT(counter);
CAN_s.Data.Databox_data_4[4] := INT_TO_USINT(counter);

IF counter = CYCLES_FOR_CAN_SEND THEN
	counter	:= 0;
	IF CAN_s.Status.Channel_CAN_1 <> 0 THEN
		can_start(CAN_1);
	END_IF
END_IF
CASE counter OF
	0:	can_sendDatabox(CAN_1, 3, 8, ADR(CAN_s.Data.Databox_data_1) );
	1:	can_sendDatabox(CAN_2, 3, 8, ADR(CAN_s.Data.Databox_data_2) );
	2: can_sendDatabox(CAN_3, 3, 8, ADR(CAN_s.Data.Databox_data_3) );
	3: can_sendDatabox(CAN_4, 3, 8, ADR(CAN_s.Data.Databox_data_4) );
	4:	;
	5:	;
	6: ;
	7:	;
	8: ;
	9: ;
	ELSE
;
END_CASE
counter	:= counter + 1;
END_ACTION
END_PROGRAM

(* POU 10_Inputs/General Parameters/Get_Dig_Freq_Inputs, ST *)
PROGRAM Get_Dig_Freq_Inputs
VAR

END_VAR
;
END_PROGRAM

(* POU Startlock_RC28_14, ST *)
(*************************************************************************************
PROGRAM: Startlock_RC28_14

BRIEF: check secure condition before starting RC 

*************************************************************************************
 (c) Copyright by BOSCH REXROTH AG, all rights reserved 
*************************************************************************************
PROJECT: DPCA40 for RC28-14/30

VERSION INFORMATION
	V1.0 	Benez Fabien, DC-MA/EMF2 (General template)
	V1.1	Lewitan Vitaly, DCRU-MA/SMC(ME2)
- errors, which are processed in this program, are configured via excell configurator
- errors can be observed via "err" structure within this application
_____________________________________________
|Best to read using Lucida Consol 9pt (Cyrillic) 	|
|tab-width=3 				             			|   	
|____________________________________________|
see  [Project] [Options] [Editor] [Fonts]
*************************************************************************************)
PROGRAM Startlock_RC28_14
VAR
	stStartlock_Condition_s16				: INT; 	(*state of the startlock*)

	uSupply_VB_mV_u16							: UINT;	(*voltage of VB*)
	uSupply_VP_1_mV_u16						: UINT;	(*voltage of VP*)
	uSupply_VSS_1_mV_u16						: UINT;	(*voltage of VSS1*)
	uSupply_VSS_2_mV_u16						: UINT;	(*voltage of VSS2*)
	uSupply_VSS_3_mV_u16						: UINT;	(*voltage of VSS3*)

	setVP_1_u16									: UINT;	(*state of the power supply1*)
	setVP_2_u16									: UINT;	(*state of the power supply2*)

	st_INH_b8									: BOOL; 	(*state of the inhibit pin*)

	stError_Case_u16							: UINT;	(*consequence of the errors: LIMP home, Stop, Ignored...*)
	Counter_s16									: INT;	(* counter for the activation of the error-reaction*)

	stSafoutCableBrake_b8					: BOOL; 	(* TRUE if no cable brake detection*)
	stSafoutShortCircuit_b8					: BOOL;	(* TRUE if no short circuit detection*)
	stSafoutFinished_b8						: BOOL;	(* TRUE if the Safout check is done*)

	Mo_ErrorCheck_Empty_b8					: BOOL;

	fb_ERR_PWRON_supply_vb_low			: handleError; (* error detection by start- vb_low*)
	fb_ERR_PWRON_supply_vss				: handleError; (* error detection by start- supply_vss*)
	fb_ERR_PWRON_hwmonitor_1				: handleError; (* error detection by start- hwmonitor_1*)
	fb_ERR_PWRON_startcondition_1		: handleError; (* error detection by start- startcondition_1*)
	fb_ERR_PWRON_engine_speed			: handleError; (* error detection by start- engine_speed*)
	fb_ERR_PWRON_hwmonitor_2				: handleError; (* error detection by start- hwmonitor_2*)
	fb_ERR_PWRON_startcondition_2		: handleError; (* error detection by start- startcondition_2*)
	fb_ERR_PWRON_safout_cable_brake	: handleError; (* error detection by start- safout_cable_brake*)
	fb_ERR_PWRON_safout_short_circuit	: handleError; (* error detection by start- safout_short_circuit*)
	fb_ERR_PWRON_powerswitch_1			: handleError; (* error detection by start- powerswitch_1*)
	fb_ERR_PWRON_powersupply				: handleError; (* error detection by start- powersupply*)
	fb_ERR_PWRON_powerswitch_2			: handleError; (* error detection by start- powerswitch_2*)
	fb_ERR_PWRON_reverse_power			: handleError; (* error detection by start- reverse_power*)
	fb_ERR_PWRON_emergency_stopp		: handleError; (* error detection by start- emergency_stop*)

(*  	stError_case_au16: ARRAY [0..20] OF UINT;   *)

	stSafout_PumpL_u16: UINT;
	stSafout_PumpR_u16: UINT;
	safout_L_s: safout_ts;
	safout_R_s: safout_ts;
	stError_case_au16: ARRAY [0..20] OF UINT;
END_VAR

VAR_INPUT
	StartconditionAppl_I_b8			: BOOL;	(* first start condition defined by the user*)
	StartconditionAppl_II_b8		: BOOL;	(* second start condition defined by the used*)
	StartconditionEngine_b8			: BOOL;	(* condition on the diesel to start the vehicle*)
	EnableSafout_b8							: BOOL;	(* defines if the safout part should be active or not*)

	tiCycle_s16									: INT;	(* cycle time of the start block*)
END_VAR

VAR_OUTPUT
	StartEnable_b8							: BOOL; 	(*TRUE is the start block has detected no error*)
	Mo_ErrorCheck_Ignore_b8			: BOOL;	(*TRUE if there is an monitor-error and if it should be ignored*)
	Mo_ErrorCheck_LimpHome_b8		: BOOL;	(*TRUE if there is an monitor-error and if the LIMP home is required*)
	Mo_ErrorCheck_Stop_b8				: BOOL;	(*TRUE if there is an monitor-error and if the vehicle has to stop*)
	Mo_ErrorCheck_Switch_b8			: BOOL; 	(*TRUE if there is an monitor-error and if the switches should be down*)
	stCase_u16									: INT; 	(*state of the start block*)
 END_VAR

VAR CONSTANT
	STARTLOCK_CHECK_SUPPLY_VB_DS16				: INT		:= 0;
	STARTLOCK_CHECK_SUPPLY_VSS_DS16				: INT		:= 1;
	STARTLOCK_READ_HWMONITOR_1_DS16				: INT		:= 2;
	STARTLOCK_CHECK_HWMONITOR_1_DS16			: INT		:= 3;
	STARTLOCK_CHECK_CONDITION_1_DS16			: INT		:= 4;
	STARTLOCK_CHECK_SWITCH_DS16						: INT		:= 5;
	STARTLOCK_CONFIG_SAFOUT_DS16					: INT		:= 6;
	STARTLOCK_CHECK_SAFOUT_DS16						: INT		:= 7;
	STARTLOCK_CHECK_ENGINE_SPEED_DS16			: INT		:= 8;
	STARTLOCK_CONFIG_VSS_DS16							: INT		:= 9;
	STARTLOCK_READ_HWMONITOR_2_DS16				: INT		:= 10;
	STARTLOCK_CHECK_HWMONITOR_2_DS16			: INT		:= 11;
	STARTLOCK_CHECK_CONDITION_2_DS16			: INT		:= 12;
	STARTLOCK_RUN_DS16										: INT		:= 13;

	ERROR_NO_DU16													: UINT	:= 0;

	ERROR_DELAY_DU16											: UINT	:= 400; (* max. known delay time is the time for config safout channels- spec. to 200ms*)

END_VAR
(************************************************************************************)
(******************** Read values for the FSM  **************************************)
(************************************************************************************)

(******************)
(** SUPPLY: VB/VP *)
(******************)
		uSupply_VB_mV_u16			:= sys_getSupply(VB);    (* Battary Voltage *)
		uSupply_VP_1_mV_u16		:= sys_getSupply(VP_1); (* Prop. Power Supply Voltage *)

(*****************)
(** SUPPLY: VSSx *)
(*****************)
		uSupply_VSS_1_mV_u16	:= sys_getSupply(VSS_1);   (* Sensor Supply *)
		uSupply_VSS_2_mV_u16	:= sys_getSupply(VSS_2);
		uSupply_VSS_3_mV_u16	:= sys_getSupply(VSS_3);

(*********************)
(* check VP switches *)
(*********************)
		(* see in state *)

(***********************)
(* check inhibit state *)
(***********************)
		st_INH_b8							:= USINT_TO_BOOL(sys_getINH());

(***************************)
(* check safout conditions *)
(***************************)
		(* see action safout status *)

(****************************************)
(* check start conditions of application*)
(****************************************)

(************************************************************************************)
(******************** FSM  **********************************************************)
(************************************************************************************)
(* check secure condition before starting RC to operate *)
CASE stStartlock_Condition_s16 OF

(*1- check Vb supply>8.5V*)
STARTLOCK_CHECK_SUPPLY_VB_DS16:
		(* startcondition flag *)
		StartEnable_b8	:= FALSE;
		(* transition *)
		IF (uSupply_VB_mV_u16 > 8500) THEN
			stStartlock_Condition_s16 := STARTLOCK_CHECK_SUPPLY_VSS_DS16;
		ELSE
			;
		END_IF

(*2- check Vssx>threshold*)
STARTLOCK_CHECK_SUPPLY_VSS_DS16:
		(* startcondition flag *)
		StartEnable_b8	:= FALSE;
		(* transition *)
		IF (
			(uSupply_VSS_1_mV_u16 > 4500) AND
			(*(uSupply_VSS_2_mV_u16 > 9500) AND*)
			(uSupply_VSS_3_mV_u16 > 4500)
			) THEN
			stStartlock_Condition_s16	:= STARTLOCK_READ_HWMONITOR_1_DS16;
		ELSE
			;
		END_IF

(*3- read HW monitor1*)
STARTLOCK_READ_HWMONITOR_1_DS16:
		(* startcondition flag *)
		StartEnable_b8	:= FALSE;
		(* do *)
		(* read hardware monitor *)
		Startlock_RC28_14.monitor_status();

		(* transition *)
		stStartlock_Condition_s16	:= STARTLOCK_CHECK_HWMONITOR_1_DS16;

(*4- check HW monitor1*)
STARTLOCK_CHECK_HWMONITOR_1_DS16:
		(* startcondition flag *)
		StartEnable_b8	:= FALSE;
		(* transition *)
		IF (Mo_ErrorCheck_Stop_b8 = FALSE AND Mo_ErrorCheck_Switch_b8 = FALSE) THEN
			stStartlock_Condition_s16	:= STARTLOCK_CHECK_CONDITION_1_DS16;
		ELSE
			;
		END_IF

(*5- check application specific start condition 1*)
STARTLOCK_CHECK_CONDITION_1_DS16:
		(* startcondition flag *)
		StartEnable_b8	:= FALSE;
		(* transition *)
		IF (StartconditionAppl_I_b8 = TRUE) THEN
			stStartlock_Condition_s16	:= STARTLOCK_CHECK_SWITCH_DS16;
		ELSE
			;
		END_IF

(*6- close central switch and check status*)
STARTLOCK_CHECK_SWITCH_DS16:
		(* startcondition flag *)
		StartEnable_b8	:= FALSE;
		(* do *)
		setVP_1_u16	:= sys_setVP( VP_1, ON );				(* PWM-supply *)
		setVP_2_u16	:= sys_setVP( VP_2, ON );				(* DIGout-supply *)
		(* transition *)
		IF (setVP_1_u16 = 16#0000 AND setVP_2_u16 = 16#0000) THEN

			Startlock_RC28_14.CAN_Status(); (* Reset each CAN line in case of shut dn *)

			IF (EnableSafout_b8 = TRUE) THEN
				stStartlock_Condition_s16	:= STARTLOCK_CONFIG_SAFOUT_DS16;
			ELSE
				stStartlock_Condition_s16	:= STARTLOCK_CHECK_ENGINE_SPEED_DS16;
			END_IF
		ELSE
			;
		END_IF

(*7- config safout channels*)
STARTLOCK_CONFIG_SAFOUT_DS16:
		(* startcondition flag *)
		StartEnable_b8	:= FALSE;
		(* optional SAFOUT Lib for customer *)
		(* do *)
		Startlock_RC28_14.safout_init();
		(* transition *)
		stStartlock_Condition_s16	:= STARTLOCK_CHECK_SAFOUT_DS16;

(*8- check for successful configuration*)
STARTLOCK_CHECK_SAFOUT_DS16:
		(* startcondition flag *)
		StartEnable_b8	:= FALSE;
		(* do *)
		Startlock_RC28_14.safout_status();

		IF (stSafoutCableBrake_b8 = TRUE OR stSafoutShortCircuit_b8 = TRUE) THEN
			Mo_ErrorCheck_LimpHome_b8	:= TRUE;
		ELSE
			;
		END_IF

		(* transition *)
		IF (stSafoutFinished_b8 = TRUE) THEN
			stStartlock_Condition_s16	:= STARTLOCK_CHECK_ENGINE_SPEED_DS16;
		ELSE
			;
		END_IF

(*9- check diesel engine speed > threshold*)
STARTLOCK_CHECK_ENGINE_SPEED_DS16:
		(* startcondition flag *)
		StartEnable_b8	:= FALSE;
		(* transition *)
		IF (StartconditionEngine_b8 = TRUE) THEN
			stStartlock_Condition_s16	:= STARTLOCK_CONFIG_VSS_DS16;
		ELSE
			;
		END_IF

(*10- config VSS1-3 Monitor*)
STARTLOCK_CONFIG_VSS_DS16:
		(* startcondition flag *)
		StartEnable_b8	:= FALSE;
		(* do *)
		mo_cfgCheck(MO_VSS_1, MO_CHECK_ON);
		mo_cfgCheck(MO_VSS_2, MO_CHECK_ON);
		mo_cfgCheck(MO_VSS_3, MO_CHECK_ON);
		(* transition *)
		stStartlock_Condition_s16	:= STARTLOCK_READ_HWMONITOR_2_DS16;

(*11- read HW monitor2*)
STARTLOCK_READ_HWMONITOR_2_DS16:
	(* startcondition flag *)
		StartEnable_b8	:= FALSE;
	(* do *)
	(* read hardware monitor *)
		Startlock_RC28_14.monitor_status();
	(* transition *)
		stStartlock_Condition_s16	:= STARTLOCK_CHECK_HWMONITOR_2_DS16;

(*12- Check HW monitor2*)
STARTLOCK_CHECK_HWMONITOR_2_DS16:
		(* startcondition flag *)
		StartEnable_b8	:= FALSE;
		(* transition *)

		IF (Mo_ErrorCheck_Stop_b8 = FALSE AND Mo_ErrorCheck_Switch_b8 = FALSE) THEN
			stStartlock_Condition_s16	:= STARTLOCK_CHECK_CONDITION_2_DS16;
		ELSE
			;
		END_IF


(*13- check application specific start condition 2*)
STARTLOCK_CHECK_CONDITION_2_DS16:
		(* startcondition flag *)
		StartEnable_b8	:= FALSE;
		(* transition *)
		IF (StartconditionAppl_II_b8 = TRUE) THEN
			stStartlock_Condition_s16	:= STARTLOCK_RUN_DS16;
		ELSE
			;
		END_IF

(*13- RUN*)
STARTLOCK_RUN_DS16:
		(* startcondition flag *)
		StartEnable_b8	:= TRUE;
		(* do customer application *)
			;

ELSE
	(* this state should never be reached *)
	stStartlock_Condition_s16 := STARTLOCK_CHECK_SUPPLY_VSS_DS16;
END_CASE

stCase_u16 := stStartlock_Condition_s16;


(*************************************************************************************************************)
(******************** ERROR - STARTBLOC **********************************************************************)
(*************************************************************************************************************)

(*********************************************)
(******** @ERR: CHECK_SUPPLY *****************)
(*********************************************)
	fb_ERR_PWRON_supply_vb_low(
					stErrorCondition_b8	:= (stStartlock_Condition_s16 = STARTLOCK_CHECK_SUPPLY_VB_DS16),
					stQuitCondition_b8	:= TRUE,
					tiDelay_u16				:= ERROR_DELAY_DU16,
					numErr_code_u16		:= ERR_PWRON_SUPPLY_VB_LOW,
					numErr_nbr_u8			:= 0,
					bSave_b8					:= FALSE,
					tiCycle_s16				:= tiCycle_s16,
					bFlag_b8					=> err.Pwron_supply_vb_low_b8);


(*********************************************)
(******** @ERR: CHECK_VSS ********************)
(*********************************************)
	fb_ERR_PWRON_supply_vss(
					stErrorCondition_b8	:= (stStartlock_Condition_s16 = STARTLOCK_CHECK_SUPPLY_VSS_DS16),
					stQuitCondition_b8	:= TRUE,
					tiDelay_u16				:= ERROR_DELAY_DU16,
					numErr_code_u16		:= ERR_PWRON_SUPPLY_VSS,
					numErr_nbr_u8			:= 0,
					bSave_b8					:= TRUE,
					tiCycle_s16				:= tiCycle_s16,
					bFlag_b8					=> err.Pwron_supply_vss_b8);

(*********************************************)
(******** @ERR: CHECK_HWMONITOR1**************)
(*********************************************)
	fb_ERR_PWRON_hwmonitor_1(
					stErrorCondition_b8	:= (stStartlock_Condition_s16 = STARTLOCK_CHECK_HWMONITOR_1_DS16),
					stQuitCondition_b8	:= TRUE,
					tiDelay_u16				:= ERROR_DELAY_DU16,
					numErr_code_u16		:= ERR_PWRON_HWMONITOR_1,
					numErr_nbr_u8			:= 0,
					bSave_b8					:= TRUE,
					tiCycle_s16				:= tiCycle_s16,
					bFlag_b8					=> err.Pwron_hwmonitor_1_b8);

(*********************************************)
(******** @ERR: CHECK_CONDITION_1 ************)
(*********************************************)
	fb_ERR_PWRON_startcondition_1(
					stErrorCondition_b8	:= (stStartlock_Condition_s16 = STARTLOCK_CHECK_CONDITION_1_DS16),
					stQuitCondition_b8	:= TRUE,
					tiDelay_u16				:= ERROR_DELAY_DU16,
					numErr_code_u16		:= ERR_PWRON_STARTCONDITION_1,
					numErr_nbr_u8			:= 0,
					bSave_b8					:= FALSE,
					tiCycle_s16				:= tiCycle_s16,
					bFlag_b8					=> err.Pwron_startcondition_1_b8);

(*********************************************)
(******** @ERR: CHECK_DIESELSPEED ************)
(*********************************************)
	fb_ERR_PWRON_engine_speed(
					stErrorCondition_b8	:= (stStartlock_Condition_s16 = STARTLOCK_CHECK_ENGINE_SPEED_DS16),
					stQuitCondition_b8	:= TRUE,
					tiDelay_u16				:= ERROR_DELAY_DU16,
					numErr_code_u16		:= ERR_PWRON_ENGINE_SPEED,
					numErr_nbr_u8			:= 0,
					bSave_b8					:= FALSE,
					tiCycle_s16				:= tiCycle_s16,
					bFlag_b8					=> err.Pwron_engine_speed_b8);

(*********************************************)
(******** @ERR: CHECK_HWMONITOR2**************)
(*********************************************)
	fb_ERR_PWRON_hwmonitor_2(
					stErrorCondition_b8	:= (stStartlock_Condition_s16 = STARTLOCK_CHECK_HWMONITOR_2_DS16),
					stQuitCondition_b8	:= TRUE,
					tiDelay_u16				:= ERROR_DELAY_DU16,
					numErr_code_u16		:= ERR_PWRON_HWMONITOR_2,
					numErr_nbr_u8			:= 0,
					bSave_b8					:= TRUE,
					tiCycle_s16				:= tiCycle_s16,
					bFlag_b8					=> err.Pwron_hwmonitor_2_b8);

(*********************************************)
(******** @ERR: CHECK_CONDITION_2 ************)
(*********************************************)
	fb_ERR_PWRON_startcondition_2(
					stErrorCondition_b8	:= (stStartlock_Condition_s16 = STARTLOCK_CHECK_CONDITION_2_DS16),
					stQuitCondition_b8	:= TRUE,
					tiDelay_u16				:= ERROR_DELAY_DU16,
					numErr_code_u16		:= ERR_PWRON_STARTCONDITION_2,
					numErr_nbr_u8			:= 0,
					bSave_b8					:= FALSE,
					tiCycle_s16				:= tiCycle_s16,
					bFlag_b8					=> err.Pwron_startcondition_2_b8);

(*********************************************)
(******** @ERR: CHECK_SAFOUT - cable_brake ***)
(*********************************************)
	fb_ERR_PWRON_safout_cable_brake(
					stErrorCondition_b8	:= (stSafoutCableBrake_b8	= TRUE),
					stQuitCondition_b8	:= TRUE,
					tiDelay_u16				:= ERROR_DELAY_DU16,
					numErr_code_u16		:= ERR_PWRON_SAFOUT_CABLE_BRAKE,
					numErr_nbr_u8			:= 0,
					bSave_b8					:= TRUE,
					tiCycle_s16				:= tiCycle_s16,
					bFlag_b8					=> err.Pwron_safout_cable_brake_b8);

(*********************************************)
(******** @ERR:CHECK_SAFOUT - short_circuit***)
(*********************************************)
	fb_ERR_PWRON_safout_short_circuit(
					stErrorCondition_b8	:= (stSafoutShortCircuit_b8	= TRUE),
					stQuitCondition_b8	:= TRUE,
					tiDelay_u16				:= ERROR_DELAY_DU16,
					numErr_code_u16		:= ERR_PWRON_SAFOUT_SHORT_CIRCUIT,
					numErr_nbr_u8			:= 0,
					bSave_b8					:= TRUE,
					tiCycle_s16				:= tiCycle_s16,
					bFlag_b8					=> err.Pwron_safout_short_circuit_b8);


(*********************************************)
(******** @ERR: SWITCH - Powerswitch_1 *******)
(*********************************************)
	fb_ERR_PWRON_powerswitch_1(
					stErrorCondition_b8	:= (
						(stStartlock_Condition_s16 = STARTLOCK_CHECK_SWITCH_DS16)  AND
	(setVP_1_u16 = SYSSETVP_ON_LOCKED_DU16 OR setVP_2_u16 = SYSSETVP_ON_LOCKED_DU16)
																					),
					stQuitCondition_b8	:= TRUE,
					tiDelay_u16				:= ERROR_DELAY_DU16,
					numErr_code_u16		:= ERR_PWRON_POWERSWITCH_1,
					numErr_nbr_u8			:= 0,
					bSave_b8					:= TRUE,
					tiCycle_s16				:= tiCycle_s16,
					bFlag_b8					=> err.Pwron_powerswitch_1_b8);

(*********************************************)
(******** @ERR: SWITCH - No_power_supply *****)
(*********************************************)
	fb_ERR_PWRON_powersupply(
					stErrorCondition_b8	:= (
					(stStartlock_Condition_s16 = STARTLOCK_CHECK_SWITCH_DS16)  AND
		(setVP_1_u16 = SYSSETVP_NOUBATT_DU16 OR setVP_2_u16 = SYSSETVP_NOUBATT_DU16)
																					),
					stQuitCondition_b8	:= TRUE,
					tiDelay_u16				:= ERROR_DELAY_DU16,
					numErr_code_u16		:= ERR_PWRON_POWERSUPPLY,
					numErr_nbr_u8			:= 0,
					bSave_b8					:= FALSE,
					tiCycle_s16				:= tiCycle_s16,
					bFlag_b8					=> err.Pwron_powersupply_b8);

(*********************************************)
(******** @ERR: SWITCH - Powerswitch_2 *******)
(*********************************************)
	fb_ERR_PWRON_powerswitch_2(
					stErrorCondition_b8	:= (
					(stStartlock_Condition_s16 = STARTLOCK_CHECK_SWITCH_DS16)  AND
					(setVP_1_u16 = SYSSETVP_NOVP_DU16 OR setVP_2_u16 = SYSSETVP_NOVP_DU16)
																					),
					stQuitCondition_b8	:= TRUE,
					tiDelay_u16				:= ERROR_DELAY_DU16,
					numErr_code_u16		:= ERR_PWRON_POWERSWITCH_2,
					numErr_nbr_u8			:= 0,
					bSave_b8					:= TRUE,
					tiCycle_s16				:= tiCycle_s16,
					bFlag_b8					=> err.Pwron_powerswitch_2_b8);

(*********************************************)
(******** @ERR: SWITCH - Reverse_power  ******)
(*********************************************)
	fb_ERR_PWRON_reverse_power(

					stErrorCondition_b8	:= (
					(stStartlock_Condition_s16 = STARTLOCK_CHECK_SWITCH_DS16)  AND
(setVP_1_u16=SYSSETVP_UNEXPECTED_VP_DU16 OR setVP_2_u16 = SYSSETVP_UNEXPECTED_VP_DU16)
								),
					stQuitCondition_b8	:= TRUE,
					tiDelay_u16				:= ERROR_DELAY_DU16,
					numErr_code_u16		:= ERR_PWRON_REVERSE_POWER,
					numErr_nbr_u8			:= 0,
					bSave_b8					:= TRUE,
					tiCycle_s16				:= tiCycle_s16,
					bFlag_b8					=> err.Pwron_reverse_power_b8);


(*********************************************)
(******** @ERR: SWITCH - EMCY_stop_active  ***)
(*********************************************)
	fb_ERR_PWRON_emergency_stopp(

					stErrorCondition_b8	:= (
						(stStartlock_Condition_s16 = STARTLOCK_CHECK_SWITCH_DS16)  AND
	(setVP_1_u16 = SYSSETVP_INH_ACTIVE_DU16 OR setVP_2_u16 = SYSSETVP_INH_ACTIVE_DU16)
							),
					stQuitCondition_b8	:= TRUE,
					tiDelay_u16				:= ERROR_DELAY_DU16,
					numErr_code_u16		:= ERR_PWRON_EMERGENCY_STOP,
					numErr_nbr_u8			:= 0,
					bSave_b8					:= TRUE,
					tiCycle_s16				:= tiCycle_s16,
					bFlag_b8					=> err.Pwron_emergency_stop_b8);
END_PROGRAM
ACTION CAN_status:
(* check if a "BusOff" is occured for CAN2,CAN3 and CAN4  *)

(*
  CAN4_Status_u16 := can_getStatus(CAN_4);

  	IF (	0 <> CAN4_Status_u16 )	THEN
		can_init(CAN_4, BAUD_250K);
	END_IF
*)

;
END_ACTION
ACTION monitor_status:
	(* reset variables *)
	Counter_s16			:= 0;
	stError_Case_u16	:= 16#FF;
	(* reset error reply *)
		mo_resetErrorReply();

	WHILE(stError_Case_u16 <> 0 AND Counter_s16 <= 20) DO
			Counter_s16			:= Counter_s16 + 1;
			stError_Case_u16	:= mo_getError();
			stError_case_au16[ Counter_s16 ] := stError_Case_u16; (* VL 28/04-2012,  In order to find definite error *)

			CASE stError_Case_u16 OF
				(* no error *)
				ERROR_NO_DU16:
					Mo_ErrorCheck_Empty_b8		:= TRUE;

(* ignore errors (эти ошибки не приведут к запрету на выполнение основного ПО *)
				MOF_V12V_DU16,
				MOF_VREF_DU16,
				MOC_ROM_SINGLEBITERR_DU16,
				MOF_OP_HOURS_LIMIT_DU16:
					Mo_ErrorCheck_Ignore_b8		:= TRUE;

(* limp home errors (эти ошибки не приведут к запрету на выполнение основного ПО *)
				MOF_VSS_1_DU16,
				MOF_VSS_2_DU16,
				MOF_VSS_3_DU16,
				MOF_TEMPHW_WARNING_DU16:
					Mo_ErrorCheck_LimpHome_b8	:= TRUE;

(* stop errors (эти ошибки запретят выполнение основного ПО *)
				MOF_TEMPHW_ERROR_DU16,
				MOC_RAM_CONTENT_ERROR_DU16,
				MOC_RAM_NOT_WRITABLE_DU16,
				MOC_WDA_THRESHOLD_VIOLATION_DU16,
				MOC_GNRL_UNDEFINED_STATE_DU16,
				MOC_ROM_DOUBLEBITERR_DU16,
				MOC_COM_SPI_MALFUNCTION_DU16,
				MOC_PCP_CHECKSUMERR_DU16,
				MOC_GPTA_TIMERERR_DU16,
				MOF_VREF_PRE_EXIST_DU16,
				MOF_V12V_PRE_EXIST_DU16,
				MOF_VP_CUTOFF_3V3_DU16,
				MOF_VP_CUTOFF_1V5_DU16,
				MOF_VP_CUTOFF_SYSSETVP_DU16,
				MOF_VP_CUTOFF_CPLD_DU16,
				MOF_MM_STARTUP_DU16,
				MOF_MM_SET_RESP_TIME_DU16,
				MOF_EEPPAGE_SYSTEM_DU16,
				MOF_EEPPAGE_API_DU16,
				MOF_EEP_PRE_EXIST_DEFECTS_DU16,
				MOF_EEPPAGE_ERRORS_DU16,
				MOF_EEPPAGE_APPLICATION_DU16:
					Mo_ErrorCheck_Stop_b8		:= TRUE;

(* switch errors (эти ошибка запретит выполнение основного ПО*)
				MOF_V3V3_EXT_DU16:
					Mo_ErrorCheck_Switch_b8		:= TRUE;

			ELSE
				(* this state should never be reached *)
				Mo_ErrorCheck_Stop_b8			:= TRUE;
			END_CASE
	END_WHILE
END_ACTION
ACTION safout_init:
(* configure safety output channels *)
(*
  safout_cfg(
							UDINT_TO_UINT(IO_Chnl.SAFOUT_PUMP_L),
							IO_Chnl.POH_PUMP_FORW_L,
							IO_Chnl.POH_PUMP_REV_L,
							0, 0, DEBOUNCE_FOR_SAVOUT, FALSE);

  safout_cfg(
							UDINT_TO_UINT(IO_Chnl.SAFOUT_PUMP_R),
							IO_Chnl.POH_PUMP_FORW_R,
							IO_Chnl.POH_PUMP_REV_R,
							0, 0, DEBOUNCE_FOR_SAVOUT, FALSE);
*)
(*
safout_ignoreError(IO_Chnl.SAFOUT_PUMP_L);
safout_ignoreError(IO_Chnl.SAFOUT_PUMP_R);
*)
(*
This function disables not only outs deactivation, but error indication also, so it is not useful
*)

(* VL, 25/05-2012: Pinging is off - because I need in case of "Forward" error - to be able to use Reverse solenoids.
But as soon as I use the same safout channel for Forw and Reverse - the exsisting error will not to make possible 
to activate opposite direction solenoid. One error exists - both solenoids are off. 

There is a possibility of limited availability - needed to be checked!!! *)
;
END_ACTION
ACTION safout_status:
(* check status of safout configuration *)
	(*
	0x00 	Full availability							-> FULL_AVAILABILITY_DU8
	0x01 	Limited availability						-> LIMITED_AVAILABILITY_DU8
	0x02 	No availability							-> NO_AVAILABILITY_DU8
	0x10 	Max current limit exceeded				-> CURRENT_TIMEOUT_DU8
	0x20 	Shut down test yet not finished		-> SHUT_DOWN_TEST_DU8
	0x40 	Pinging is activ							-> PINGING_DU8
	*)

	(* set error flag for cable brake *)
(*
stSafout_PumpL_u16 := safout_getStatusxt(IO_Chnl.SAFOUT_PUMP_L, ADR(safout_L_s));
stSafout_PumpR_u16 := safout_getStatusxt(IO_Chnl.SAFOUT_PUMP_R, ADR(safout_R_s));
*)
(*
	IF (
		( stSafout_PumpL_u16 = CURRENT_TIMEOUT_DU8) OR
		(...)
		)THEN
		stSafoutCableBrake_b8 	:= TRUE;
	ELSE
		;
	END_IF
*)

	(* set error flag for short circuit *)
(*
	IF (
		(safout_getStatus(SAFOUT_37_POH) = SHUT_DOWN_TEST_DU8) OR
		(...)
		)THEN
		stSafoutShortCircuit_b8	:= TRUE;
	ELSE
		;
	END_IF  *)


	(* set flag for safout check finished *)

	IF ((* TR VL 25/05-2012 - I think - there is wrong PINGING constant in the current API -
																			a real pinging status is 16#20!!!    *)
	(stSafout_PumpL_u16 = FULL_AVAILABILITY_DU8 OR stSafout_PumpL_u16 = 16#20(*PINGING_DU8*) ) AND
	(stSafout_PumpR_u16 = FULL_AVAILABILITY_DU8 OR stSafout_PumpR_u16 = 16#20(*PINGING_DU8*) )
		) THEN
		stSafoutFinished_b8	:= TRUE;
	ELSE
		stSafoutFinished_b8	:= FALSE;
	END_IF
END_ACTION

(* POU 60_Error handling/handleError, ST *)
(*************************************************************************************
FUNCTION BLOCK: fb_handleError

BRIEF: set/reset an error under BODAS-service after a defined debounce time 

PARAM[IN]	stErrorCondition_b8  error condition						[0/1]
PARAM[IN]	stQuitCondition_b8	quit condition							[0/1]
PARAM[IN]	tiDelay_u16	 			delay time for error detection 	[ms]
PARAM[IN]	numErr_code_u16 		error code under BODAS-service	
PARAM[IN]	numErr_nbr_u8	 		error number under BODAS-service
PARAM[IN]	bSave_b8		 			1: the error is saved in EEPROM	[0/1]
PARAM[IN]	tiCycle_s16	 			cycle time

PARAM[OUT]	bFlag_b8					error currently active or not  	[0/1]

*************************************************************************************
 (c) Copyright by BOSCH REXROTH AG, all rights reserved 
*************************************************************************************

VERSION INFORMATION
	V1.0 	Benez Fabien, DC-MA/EMF2
		- initial release	
_____________________________________
|Best to read using Courrier new 8pt |
|tab-width=3 				             |   	
|____________________________________|
see  [Project] [Options] [Editor] [Fonts]
**************************************************************************************)

FUNCTION_BLOCK handleError
(*	This function block checks the error-condition and the quit-error-condition.
	If the error-condition is true for the defined time, the error is saved in the bb3-array and the error flag is set. 
	If the quit-error-condition is true, the error is deleted in the bb3-array and the error flag is reset.
*)

VAR_INPUT
	stErrorCondition_b8	: BOOL;					(* error condition *)
	stQuitCondition_b8	: BOOL	:= FALSE;	(* quit condition *)
	tiDelay_u16				: UINT	:= 0;			(* delay time for error detection  *)
	numErr_code_u16		: UINT;					(* error code under BODAS-service*)
	numErr_nbr_u8			: USINT;					(* error number under BODAS-service*)
	bSave_b8					: BOOL;					(* 1: the error is saved in EEPROM	*)
	tiCycle_s16				: INT;					(* cycle time*)
END_VAR


VAR
	cnt_s16					: INT;
END_VAR


VAR_OUTPUT
	bFlag_b8					: BOOL	:= FALSE;	(* error bit that is set in case of error *)
END_VAR
(*debouncing*)
IF stErrorCondition_b8 THEN
	cnt_s16	:= cnt_s16 + 1;
ELSE
	cnt_s16 	:= 0;
END_IF

(* if delay is reached set: BODAS error *)
IF ( cnt_s16 > tiDelay_u16 / tiCycle_s16 ) THEN

	(* error counter in B-s shall only be incremented once per occurrence of an error *)
	IF NOT bFlag_b8 THEN
		sys_setError( numErr_code_u16,  numErr_nbr_u8 , bSave_b8 );
	END_IF

	(*Prevent an overrun of cnt_s16 *)
	cnt_s16	:= cnt_s16  - 1;

	(*BODAS error active*)
	bFlag_b8	:= TRUE;

(* if quit condition is fulfilled: reset bb3 error *)
ELSIF stQuitCondition_b8 THEN

								(* reset bb3 error only if error is active  *)
				IF sys_testError( numErr_code_u16, numErr_nbr_u8) > 0 THEN
							sys_delActiveError( numErr_code_u16, numErr_nbr_u8 );
				END_IF

	(*BODAS error not active*)
	bFlag_b8	:= FALSE;

END_IF
END_FUNCTION_BLOCK

(* POU 60_Error handling/Process Errors/proc_Err_CAN, ST *)
PROGRAM proc_Err_CAN
VAR
	ProcessErr1_fb		: handleError;
	ProcessErr2_fb		: handleError;
	ProcessErr3_fb		: handleError;
	ProcessErr4_fb		: handleError;
	ProcessErr5_fb		: handleError;
	ProcessErr6_fb		: handleError;
	ProcessErr7_fb		: handleError;
	ProcessErr8_fb		: handleError;
	ProcessErr9_fb		: handleError;
	ProcessErr10_fb	: handleError;

	Can_Error_Ton		: TON;
	Can_reset_fb		: Can_reset;
	dataLen_u16			: UINT 					:= 8;
	error80_cond		: BOOL;
	error83_cond		: BOOL;
	error8A_cond		: BOOL;
	error90a_cond		: BOOL;
	error90b_cond		: BOOL;
END_VAR
IF stStartlock_b8 THEN
	Can_Error_Ton(in := TRUE, PT := T#1000ms);
	(* Run reset procedure in case of bus shutdown *)
	Can_reset_fb(	stCAN_BusOFF_b8	:= CAN_s.Status.BODAS_SERVICE_u16.0,
						Can_Channel_u8		:= CAN_s.Chnl.BODAS_SERVICE_u8);
END_IF

(**)
;
END_PROGRAM

(* POU 40_CAN/Can_reset, ST *)
(*************************************************************************************
FUNCTION_BLOCK: Can_reset

BRIEF: Reset of the CAN bus after a bus-off detection


PARAM[IN]	stCAN_BusOFF_b8	 				flag for the reset of the CAN bus [0/1]

*************************************************************************************
 (c) Copyright by BOSCH REXROTH AG, all rights reserved 
*************************************************************************************

VERSION INFORMATION
	V1.0 	Benez Fabien, DC-MA/EMF2
		- initial release	
_____________________________________
|Best to read using Courrier new 8pt |
|tab-width=3 				             |
|____________________________________|
see  [Project] [Options] [Editor] [Fonts]
**************************************************************************************)
FUNCTION_BLOCK Can_reset

VAR_INPUT
	stCAN_BusOFF_b8	: BOOL;			(*flag for the reset*)
	Can_Channel_u8		: BYTE;			(*channel of the CAN bus*)
END_VAR

VAR
	stCan_Reset_s16	: INT		:=0;	(*flag used for the reset of the CAN bus *)
	Can_reset_Ton		: TON;			(*TON for the reset of the CAN bus*)
END_VAR
(*if a bus off is detected, the CAN bus have to be reset *)
CASE stCan_Reset_s16 OF

CAN_RESET_STOP:
	IF ( stCAN_BusOFF_b8 = 1 ) THEN
		stCan_Reset_s16 := CAN_RESET_START;
	END_IF

CAN_RESET_START:
	can_init( 	Can_Channel_u8,
					BAUD_250K );
	stCan_Reset_s16 := CAN_RESET_WAIT;
	Can_reset_Ton(in := 0, PT := T#500ms);

CAN_RESET_WAIT:
	Can_reset_Ton(in := 1, PT := T#500ms);
	IF ( Can_reset_Ton.Q ) THEN
		stCan_Reset_s16 := CAN_RESET_STOP;
	END_IF

ELSE
	stCan_Reset_s16 := CAN_RESET_STOP;
END_CASE;
END_FUNCTION_BLOCK

(* POU 60_Error handling/flash_Error_Code, ST *)
(*************************************************************************************
* PROGRAM flash_Error_Code
*/
* Provide 2 digit flash code indication.
**************************************************************************************************
* (c) Copyright by BOSCH REXROTH AG, all rights reserved *
**************************************************************************************************
**************************************************************************************************
* PROJECT:	 Universal
* VERSION INFORMATION: 
*	v1.00, 27.03.2012, Vitaly Lewitan, DCRU-MA/SMC

* REVISION HISTORY:
* no revision so far
*
*
*)

(* insert command RETURN to deactivate this function block *)
(* RETURN; *)
PROGRAM flash_Error_Code
VAR CONSTANT
	ELC_WAIT:											INT	:= 0;
	ELC_PAUSE_10_1_PREP:			INT	:= 4;
	ELC_PAUSE_10_1:							INT	:= 5;
	ELC_PAUSE_LONG_PREP:		INT	:= 6;
	ELC_PAUSE_LONG:						INT	:= 7;
	ELC_FLASH_10_PREP:				INT	:= 8;
	ELC_FLASH_10_ON:						INT	:= 9;
	ELC_FLASH_10_OFF:					INT	:= 10;
	ELC_FLASH_1_PREP:					INT	:= 11;
	ELC_FLASH_1_ON:						INT	:= 12;
	ELC_FLASH_1_OFF:						INT	:= 13;
END_VAR
VAR
	stErrorLampControl_s16: INT := ELC_WAIT;  (* переменная статуса управления лампой ошибки *)
	Blink_Code_Digit_s16: INT;
	BlinkTimer_fb: TON;
END_VAR
VAR_INPUT
	BlinkCode_s16: INT;
	tiBlink10H_u32: TIME;
	tiBlink10L_u32: TIME;
	tiBlinkPause_10_1_u32: TIME;
	tiBlink1_H_u32: TIME;
	tiBlink1_L_u32: TIME;
	tiPauseLong_u32: TIME;
END_VAR
VAR_OUTPUT
	ErrLamp_b8: BOOL;
	Error_Indication_Completed_b8: BOOL;
END_VAR
BlinkTimer_fb;

CASE stErrorLampControl_s16 OF   (* переменная статуса процедуры управления лампой ошибки ПУЛО*)

ELC_WAIT:
		ErrLamp_b8 := FALSE;
		Error_Indication_Completed_b8 := FALSE;
 		IF BlinkCode_s16 > 0 THEN
				stErrorLampControl_s16 := ELC_FLASH_10_PREP;
		ELSE
				stErrorLampControl_s16 := ELC_WAIT;
		END_IF

ELC_FLASH_10_PREP:
		Blink_Code_Digit_s16 := BlinkCode_s16 / 10;
(*		Blink_Code_Digit_s16 := Blink_Code_Digit_s16 MOD 10;  ????????? *)
		BlinkTimer_fb( in := FALSE );
		BlinkTimer_fb.PT := tiBlink10H_u32;
		BlinkTimer_fb( in :=TRUE );
		stErrorLampControl_s16 := ELC_FLASH_10_ON;

ELC_FLASH_10_ON:     (* сигнала старшего разряда, ЛО включена *)
		IF Blink_Code_Digit_s16 <= 0 THEN
			stErrorLampControl_s16 := ELC_PAUSE_10_1_PREP;  (* порепрыгиваем на мигалку младших разрядов *)
		ELSE
			ErrLamp_b8 := TRUE;  (* включение ЛО *)

			IF BlinkTimer_fb.Q THEN
				BlinkTimer_fb( in := FALSE );
				BlinkTimer_fb.PT := tiBlink10L_u32;
				BlinkTimer_fb( in := TRUE );
				stErrorLampControl_s16 := ELC_FLASH_10_OFF;  (* Переход на сл. шаг *)
			END_IF
		END_IF

ELC_FLASH_10_OFF:
		ErrLamp_b8 := FALSE;   (* выключение ЛО *)
		IF BlinkTimer_fb.Q THEN
			BlinkTimer_fb( in := FALSE );
			BlinkTimer_fb.PT := tiBlink10H_u32;
			BlinkTimer_fb( in := TRUE );
			Blink_Code_Digit_s16 := Blink_Code_Digit_s16 - 1;  (* счётчик миганий ЛО *)
			stErrorLampControl_s16 := ELC_FLASH_10_ON;
		END_IF

ELC_PAUSE_10_1_PREP:
		BlinkTimer_fb( in := FALSE );
		BlinkTimer_fb.PT := tiBlinkPause_10_1_u32;
		BlinkTimer_fb( in :=TRUE );
		stErrorLampControl_s16 := ELC_PAUSE_10_1;

ELC_PAUSE_10_1:
		ErrLamp_b8 := FALSE;

		IF BlinkTimer_fb.Q THEN
			BlinkTimer_fb( in := FALSE );
			stErrorLampControl_s16 := ELC_FLASH_1_PREP;
		END_IF


ELC_FLASH_1_PREP:
		Blink_Code_Digit_s16 := BlinkCode_s16 MOD 10;
		BlinkTimer_fb( in := FALSE );
		BlinkTimer_fb.PT := tiBlink1_H_u32;
		BlinkTimer_fb( in := TRUE );

		stErrorLampControl_s16 := ELC_FLASH_1_ON;


ELC_FLASH_1_ON:                 (* сигнал ЛО младшего разряда, ЛО включена *)
		IF Blink_Code_Digit_s16 <= 0 THEN
			stErrorLampControl_s16 := ELC_PAUSE_LONG_PREP;
		ELSE
			ErrLamp_b8 := TRUE;     (* включение ЛО *)
					IF BlinkTimer_fb.Q THEN
						BlinkTimer_fb( in := FALSE );
						BlinkTimer_fb.PT := tiBlink1_L_u32;
						BlinkTimer_fb( in := TRUE );
						stErrorLampControl_s16 := ELC_FLASH_1_OFF;
					END_IF
		END_IF

ELC_FLASH_1_OFF:
		ErrLamp_b8 := FALSE;
		IF BlinkTimer_fb.Q THEN
			BlinkTimer_fb( in := FALSE );
			BlinkTimer_fb.PT := tiBlink1_H_u32;
			BlinkTimer_fb( in := TRUE );
			Blink_Code_Digit_s16 := Blink_Code_Digit_s16 - 1;
			stErrorLampControl_s16 := ELC_FLASH_1_ON;
		END_IF

ELC_PAUSE_LONG_PREP:
		BlinkTimer_fb( in := FALSE );
		BlinkTimer_fb.PT := tiPauseLong_u32;
		BlinkTimer_fb( in := TRUE );
		stErrorLampControl_s16 := ELC_PAUSE_LONG;

ELC_PAUSE_LONG:
		ErrLamp_b8 := FALSE;
		Error_Indication_Completed_b8 := TRUE;
		IF BlinkTimer_fb.Q THEN
			stErrorLampControl_s16 := ELC_WAIT;
		END_IF

END_CASE
END_PROGRAM

(* POU 60_Error handling/review_Errors, ST *)
(*************************************************************************************
* PROGRAM displayErrorCode
*/
* Provide cyclically changed Active or Saved error code - for i.e. indication on display or for flash code indication.
*Error codes retrieved from the RunTime system, from the "ErrorData_ts" structure.
**************************************************************************************************
**************************************************************************************************
*
**************************************************************************************************
* (c) Copyright by BOSCH REXROTH AG, all rights reserved *
**************************************************************************************************
**************************************************************************************************
Used following user defined type:

TYPE ErrorData_ts :
STRUCT
  Code_u16: UINT;   (* Error code (module + function + type). *)
  Param_u8: USINT;      (* Error parameter. *)
  Occurrence_u8: USINT;  (* Error occurrence counter. *)
  Timestamp_u32: UDINT; (* Timestamp of the last occurrence in minutes (value of the operating time counter). *)
END_STRUCT
END_TYPE
***************************************************************************************************
***************************************************************************************************
* PROJECT:	 Universal
* VERSION INFORMATION: 
*	v1.00, 27.03.2012, Vitaly Lewitan, DCRU-MA/SMC
*  v1.01, 03/05-2012, Vitaly Lewitan, DCRU-MA/SMC. System errors are not displayed!!!
*  v1.02, 03/05-2012, Vitaly Lewitan, DCRU-MA/SMC. Module adapted for flash code (instead of timer, 
				"error indication comlete" flag is used for switching to the next error 
* REVISION HISTORY:
* no revision so far
*
*
*)

PROGRAM review_Errors
VAR
	numErr_s16: INT;
	stErr_indication_s16: INT;
	idxError_s16: INT;
	errors_as: ARRAY [1..200] OF ErrorData_ts;
	Error_Code_u16: UINT;
	Error_Code_s16: INT;
END_VAR
VAR_OUTPUT
	Displayed_Err_Code_s16: INT;
END_VAR
VAR_INPUT
	Saved_Err_b8: BOOL;
	Last_Error_Shown_b8: BOOL;
END_VAR
VAR CONSTANT
	CHECK_FOR_ERRORS: INT := 0;
	DISPLAY_ERROR_PREP: INT := 2;
	DISPLAY_ERROR: INT := 1;
END_VAR
IF Saved_Err_b8 THEN
numErr_s16 := UINT_TO_INT(sys_getNumSavedErrors());
sys_getSavedErrors(ADR(errors_as[1]), 0, 200 );
ELSE
numErr_s16 := UINT_TO_INT(sys_getNumActiveErrors());
sys_getActiveErrors(ADR(errors_as[1]), 0, 200 );
END_IF

CASE stErr_indication_s16 OF

CHECK_FOR_ERRORS:

			IF numErr_s16 <= 0 THEN
					Displayed_Err_Code_s16 := 0;
					idxError_s16 := 0;
			ELSIF idxError_s16 >= numErr_s16 THEN (* all active errors were displayed *)
					idxError_s16 := 0;
			ELSE  (* Display the next error *)
						idxError_s16 := idxError_s16 + 1; (* Next error  *)
						Error_Code_u16 := errors_as[idxError_s16].Code_u16;
															IF Error_Code_u16 >= 16#8000  (* application error *)
																THEN
															Error_Code_s16 := UINT_TO_INT(Error_Code_u16 - 16#8000);
															stErr_indication_s16 := DISPLAY_ERROR_PREP;
															ELSE  (* system error, no indication *)
															stErr_indication_s16 := CHECK_FOR_ERRORS;
															Displayed_Err_Code_s16 := 0;
															END_IF
			END_IF

DISPLAY_ERROR_PREP:
			IF NOT Last_Error_Shown_b8 THEN (* previous error indication completed *)
				stErr_indication_s16 := DISPLAY_ERROR;
			ELSE
				stErr_indication_s16 := DISPLAY_ERROR_PREP;(* keep found error till the long pause of the prev. error completed *)
			END_IF

DISPLAY_ERROR:

   Displayed_Err_Code_s16 := Error_Code_s16;

			IF Last_Error_Shown_b8 THEN  (* indication of the current error completed, look for the next error *)
					stErr_indication_s16 := CHECK_FOR_ERRORS ;
			ELSE;
			END_IF
ELSE
  stErr_indication_s16 := CHECK_FOR_ERRORS ;
END_CASE
END_PROGRAM

(* POU 30_Outputs/out_DIG, ST *)
PROGRAM out_DIG
VAR

END_VAR
VAR CONSTANT

END_VAR
(* *)
;
END_PROGRAM

(* POU Autocode/SW_Version, ST *)
PROGRAM SW_Version 
VAR 
	SW_Git_Commit_s32	: DINT;		(* First 7 characters of the current git commit, hex *) 
	SW_Git_Hash_as8	: STRING;	(* First 7 characters of the current git commit, hex *) 
END_VAR 
(*********************************************) 
(*  DON'T MAKE ANY CHANGES TO THIS PROGRAM!! *) 
(*     FILE WAS AUTOMATICALLY GENERATED!!    *) 
(*********************************************) 
SW_Git_Commit_s32 := 16#7b0d05e;
SW_Git_Hash_as8 := '7b0d05e';
END_PROGRAM

(* POU 10_Inputs/General Parameters/get_Status, ST *)
PROGRAM get_Status
VAR

	in_as: ARRAY [1..75] OF in_ts;	(* Structure with the extended input information *)

END_VAR
  (* get infos from specified input *)

  inxt(IN_1_AIV,  	ADR(in_as[1]));
  inxt(IN_2_AIV, 		ADR(in_as[2]));
  inxt(IN_3_AIV,  	ADR(in_as[3]));
  inxt(IN_4_AIV,  	ADR(in_as[4]));
  inxt(IN_5_AIV,  	ADR(in_as[5]));
  inxt(IN_6_AIV,  	ADR(in_as[6]));
  inxt(IN_7_AIV,  	ADR(in_as[7]));
  inxt(IN_8_AIV,  	ADR(in_as[8]));
  inxt(IN_9_AIV,  	ADR(in_as[9]));
  inxt(IN_10_AIV,  	ADR(in_as[10]));
  inxt(IN_11_AIV,  	ADR(in_as[11]));
  inxt(IN_12_AIV,  	ADR(in_as[12]));
  inxt(IN_13_AIV,  	ADR(in_as[13]));
  inxt(IN_14_AIV,  	ADR(in_as[14]));
  inxt(IN_15_AIV,  	ADR(in_as[15]));
  inxt(IN_16_AIV,  	ADR(in_as[16]));
  inxt(IN_17_AIV,  	ADR(in_as[17]));
  inxt(IN_18_AIV,  	ADR(in_as[18]));
  inxt(IN_19_AIV,  	ADR(in_as[19]));
  inxt(IN_20_AIV,  	ADR(in_as[20]));
  inxt(IN_21_AIV,  	ADR(in_as[21]));
  inxt(IN_22_AIV,  	ADR(in_as[22]));
  inxt(IN_23_AIV,  	ADR(in_as[23]));
  inxt(IN_24_AIV,  	ADR(in_as[24]));
  inxt(IN_25_AIV,  	ADR(in_as[25]));
  inxt(IN_26_AIV,  	ADR(in_as[26]));
  inxt(IN_27_AIV,  	ADR(in_as[27]));
  inxt(IN_28_AIV,  	ADR(in_as[28]));
  inxt(IN_29_AIV,  	ADR(in_as[29]));
  inxt(IN_30_AIV,  	ADR(in_as[30]));
  inxt(IN_31_AIV,  	ADR(in_as[31]));
  inxt(IN_32_AIV,  	ADR(in_as[32]));
  inxt(IN_33_AIV,  	ADR(in_as[33]));
  inxt(IN_34_AIV,  	ADR(in_as[34]));
  inxt(IN_35_AIV,  	ADR(in_as[35]));
  inxt(IN_36_AIV,  	ADR(in_as[36]));
  inxt(IN_37_AIV,  	ADR(in_as[37]));
  inxt(IN_38_AIV,  	ADR(in_as[38]));
  inxt(IN_39_AIV,  	ADR(in_as[39]));
  inxt(IN_40_AIV,  	ADR(in_as[40]));
  inxt(IN_41_AIV,  	ADR(in_as[41]));
  inxt(IN_42_DI,  	ADR(in_as[42]));
  inxt(IN_43_DI,  	ADR(in_as[43]));
  inxt(IN_44_DI,  	ADR(in_as[44]));
  inxt(IN_45_DI,  	ADR(in_as[45]));
  inxt(IN_46_DI,  	ADR(in_as[46]));
  inxt(IN_47_DI,  	ADR(in_as[47]));
  inxt(IN_48_DI,  	ADR(in_as[48]));
  inxt(IN_49_DI,  	ADR(in_as[49]));
  inxt(IN_50_DI,  	ADR(in_as[50]));
  inxt(IN_51_DI,  	ADR(in_as[51]));
  inxt(IN_52_AIV,  	ADR(in_as[52]));
  inxt(IN_53_AIV,  	ADR(in_as[53]));
  inxt(IN_54_AIV,  	ADR(in_as[54]));
  inxt(IN_55_AIV,  	ADR(in_as[55]));
  inxt(IN_56_AIV,  	ADR(in_as[56]));
  inxt(IN_57_AIV,  	ADR(in_as[57]));
  inxt(IN_58_AIV,  	ADR(in_as[58]));
  inxt(IN_59_AIV,  	ADR(in_as[59]));
  inxt(IN_60_AIV,  	ADR(in_as[60]));
  inxt(IN_61_AIV,  	ADR(in_as[61]));
  inxt(IN_62_AIV,  	ADR(in_as[62]));
  inxt(IN_63_AIV,  	ADR(in_as[63]));
  inxt(IN_64_AIV,  	ADR(in_as[64]));
  inxt(IN_65_AIV,  	ADR(in_as[65]));
  inxt(IN_66_AIV,  	ADR(in_as[66]));
  inxt(IN_67_AIV,  	ADR(in_as[67]));
  inxt(IN_68_AIV,  	ADR(in_as[68]));
  inxt(IN_69_AIV,  	ADR(in_as[69]));
  inxt(IN_70_AIV,  	ADR(in_as[70]));
  inxt(IN_71_FI,  	ADR(in_as[71]));
  inxt(IN_72_FI,  	ADR(in_as[72]));
  inxt(IN_73_FI,  	ADR(in_as[73]));
  inxt(IN_74_FI,  	ADR(in_as[74]));
  inxt(IN_75_FI,  	ADR(in_as[75]));
END_PROGRAM

(* POU UDS_Task, ST *)
PROGRAM UDS_Task
VAR
	DataboxData_au8: ARRAY[1..8] OF USINT;
	DataboxNumBytes_u8: USINT;
	databoxCode: UINT;
	i: USINT;
	bufferDataSize: USINT;

	tempCanSendBuff: ARRAY[1..8] OF USINT;

	bytesTxFf: ARRAY[1..8] OF USINT;
	bytesTxCf: ARRAY[1..8] OF USINT;
	startIndex: USINT;
	txCfIdx: USINT;

	y: USINT;
END_VAR
IF (Uds_s.status = 0) THEN
	databoxCode := can_getDatabox(0, 9, ADR(DataboxData_au8), ADR(DataboxNumBytes_u8));
	IF (databoxCode <> 0) THEN
		IF (Uds_s.tester = 60000) THEN (*reset session type if there are no messages (600 = 3 seconds, 60000 = 5 minutes for debug)*)
			Uds_s.sessionType := 0;
			Uds_s.tester := 0;
		ELSE
			Uds_s.tester := Uds_s.tester + 1;
		END_IF
	ELSIF (databoxCode = 0) THEN
		IF (DataboxData_au8[1] = 16#30) THEN
			Uds_s.status := 1;
		ELSIF (DataboxData_au8[1] < 16#8) THEN
			Uds_s.UdsRx.dataSize := DataboxData_au8[1];
			i := 2;
			y := 2;
			Uds_s.UdsRx.data[1] := 0;
			FOR y := 2 TO Uds_s.UdsRx.dataSize + 1 DO
				Uds_s.UdsRx.data[y] := DataboxData_au8[i];
				i := i + 1;
				Uds_s.UdsRx.data[1] := Uds_s.UdsRx.data[1] + 1;
			END_FOR
		ELSIF (DataboxData_au8[1] = 16#10) THEN
			i := 2;
			Uds_s.UdsRx.dataSize := DataboxData_au8[i];
			i := i + 1;
			y := 2;
			Uds_s.UdsRx.data[1] := 0;
			FOR y := 2 TO 6 DO
				Uds_s.UdsRx.data[y] := DataboxData_au8[i + y - 1];
				Uds_s.UdsRx.data[1] := Uds_s.UdsRx.data[1] + 1;
			END_FOR
			Uds_s.status := 1;
			Uds_s.UdsTx.dataSize := 3;
			Uds_s.UdsTx.data[1] := 16#03;
			Uds_s.UdsTx.data[2] := 16#30;
			Uds_s.UdsTx.data[3] := 16#FF;
			Uds_s.UdsTx.data[4] := 16#0A;
		ELSIF (DataboxData_au8[1] > 16#10 AND DataboxData_au8[1] < 16#30 AND Uds_s.UdsRx.dataSize > Uds_s.UdsRx.data[1]) THEN
			bufferDataSize := Uds_s.UdsRx.data[1];
			FOR y := 2 TO 7 DO
				IF (Uds_s.UdsRx.data[1] >= Uds_s.UdsRx.dataSize) THEN
					EXIT;
				END_IF
				Uds_s.UdsRx.data[bufferDataSize + y] := DataboxData_au8[y];
				Uds_s.UdsRx.data[1] := Uds_s.UdsRx.data[1] + 1;
			END_FOR
		END_IF
		Uds_s.tester := 0;
	END_IF
END_IF

